KUKA KRL program: EPS_2_251806_MH49A_A_20260212042248.src

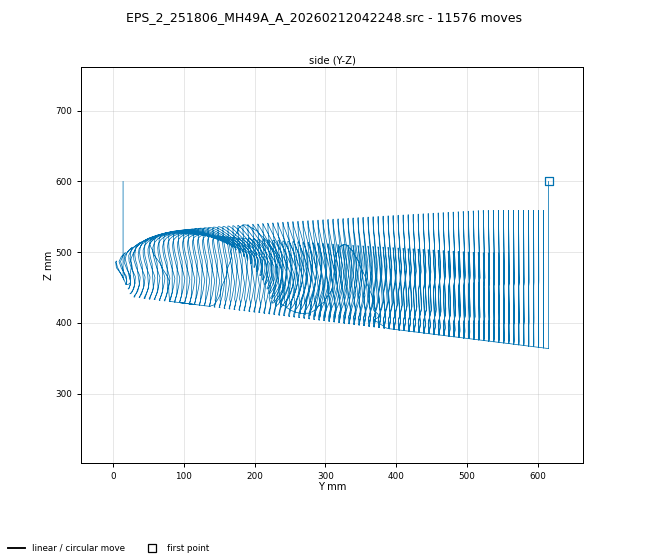
[picture p0: tool path of EPS_2_251806_MH49A_A_20260212042248.src, 11576 of 11578 moves have a stored position in this frame; points joined in program order, loops and branches not executed]
&ACCESS RVP
&REL 4
&COMMENT QRS 19112012
&PARAM EDITMASK = *
DEF PART()
EXT BAS (BAS_COMMAND :IN,REAL :IN )
INT I
BAS (#INITMOV,0 )

;KUKA QRS Post kuka4.cps  Date:22-06-2017 !

File_ID=3021

QRS_PRE_INIT()

;Init var - Until changes are made in qrs_pre_init
Outlet_Square_prg=0
Inlet_1_Square_prg=0
Inlet_2_Square_prg=0
Inlet_3_Square_prg=0
Inlet_4_Square_prg=0
Inlet_5_Square_prg=0

Outlet_1={X 0.000, Y 520.860, Z 458.500, B 0.000, E1 0.000 }
Inlet_1={X 0.000, Y 525.210, Z 398.500, B 0.000, E1 242.000 }
Outlet_1_type=201
Inlet_1_type=201
;QRS#1=Sidecore dimensions
;QRS#2=200-8" PVC SDR 35
;QRS#3=200-8" PVC SDR 35
;QRS#4=
;QRS#5=
;QRS#6=
;QRS#7=
;QRS#8=
;QRS#9=12-08 PSX
;QRS#10=12-08 PSX
;QRS#11=
;QRS#12=
;QRS#13=
;QRS#14=
;QRS#15=
;QRS#16=1220x127x838 2,75'
;QRS#17=EPS Height
;QRS#18=559
;QRS#19=*
;QRS#20= UPDATED VERSION 22-06-2017
;QRS#21=*
Outlet_Square=0100
Inlet_1_Square=0100
Inlet_2_Square=0
Inlet_3_Square=0
Inlet_4_Square=0
Inlet_5_Square=0
Mill_Square=1
Outlet_Square_Prg=204
Inlet_1_Square_prg=204

QRS_INIT()

$ADVANCE=5

; T1
PTP {E1 173.627,E2 173.627}
PTP {X 0,Y 615.485,A -85,B 0,C 180,E1 173.627,E2 173.627,E3 0,E4 0,E5 0,E6 0}
QRS_SPEED_INIT()
LIN {X 0,Y 615.485,Z 600,A -85,B 0,C 180,E1 173.627,E2 173.627,E3 0,E4 0,E5 0,E6 0} C_VEL
LIN {X 0,Y 615.485,Z 373.874,A -85,B 0,C 180,E1 173.627,E2 173.627} C_VEL
LIN {X 0,Y 615.485,Z 365.7,A -85,B 0,C 180,E1 173.627,E2 173.627} C_VEL
LIN {X 0,Y 615.471,Z 363.7,A -85,B 0,C 180,E1 173.44,E2 173.44} C_VEL
LIN {X 0,Y 615.49,Z 363.695,A -85,B 0,C 180,E1 170.802,E2 170.802} C_VEL
LIN {X 0,Y 615.467,Z 363.7,A -85,B 0,C 180,E1 168.139,E2 168.139} C_VEL
LIN {X 0,Y 615.473,Z 363.699,A -85,B 0,C 180,E1 165.451,E2 165.451} C_VEL
LIN {X 0,Y 615.485,Z 363.697,A -85,B 0,C 180,E1 162.73,E2 162.73} C_VEL
LIN {X 0,Y 615.476,Z 363.7,A -85,B 0,C 180,E1 159.968,E2 159.968} C_VEL
LIN {X 0,Y 615.494,Z 363.699,A -85,B 0,C 180,E1 157.156,E2 157.156} C_VEL
LIN {X 0,Y 615.492,Z 363.7,A -85,B 0,C 180,E1 154.285,E2 154.285} C_VEL
LIN {X 0,Y 615.492,Z 363.695,A -85,B 0,C 180,E1 151.343,E2 151.343} C_VEL
LIN {X 0,Y 615.482,Z 363.702,A -85,B 0,C 180,E1 148.916,E2 148.916} C_VEL
LIN {X 0,Y 615.483,Z 363.7,A -85,B 0,C 180,E1 146.468,E2 146.468} C_VEL
LIN {X 0,Y 615.46,Z 363.7,A -85,B 0,C 180,E1 144.171,E2 144.171} C_VEL
LIN {X 0,Y 615.483,Z 363.696,A -85,B 0,C 180,E1 141.932,E2 141.932} C_VEL
LIN {X 0,Y 615.49,Z 363.697,A -85,B 0,C 180,E1 139.395,E2 139.395} C_VEL
LIN {X 0,Y 615.481,Z 363.7,A -85,B 0,C 180,E1 136.756,E2 136.756} C_VEL
LIN {X 0,Y 615.489,Z 363.697,A -85,B 0,C 180,E1 133.999,E2 133.999} C_VEL
LIN {X 0,Y 615.464,Z 363.699,A -85,B 0,C 180,E1 131.093,E2 131.093} C_VEL
LIN {X 0,Y 615.493,Z 363.701,A -85,B 0,C 180,E1 128.906,E2 128.906} C_VEL
LIN {X 0,Y 615.492,Z 363.694,A -85,B 0,C 180,E1 125.836,E2 125.836} C_VEL
LIN {X 0,Y 615.472,Z 363.7,A -85,B 0,C 180,E1 123.239,E2 123.239} C_VEL
LIN {X 0,Y 615.495,Z 363.699,A -85,B 0,C 180,E1 120.921,E2 120.921} C_VEL
LIN {X 0,Y 615.472,Z 363.7,A -85,B 0,C 180,E1 118.449,E2 118.449} C_VEL
LIN {X 0,Y 615.499,Z 363.698,A -85,B 0,C 180,E1 115.573,E2 115.573} C_VEL
LIN {X 0,Y 615.488,Z 363.701,A -85,B 0,C 180,E1 112.846,E2 112.846} C_VEL
LIN {X 0,Y 615.494,Z 363.699,A -85,B 0,C 180,E1 110.034,E2 110.034} C_VEL
LIN {X 0,Y 615.483,Z 363.7,A -85,B 0,C 180,E1 107.273,E2 107.273} C_VEL
LIN {X 0,Y 615.483,Z 363.699,A -85,B 0,C 180,E1 104.551,E2 104.551} C_VEL
LIN {X 0,Y 615.49,Z 363.697,A -85,B 0,C 180,E1 101.863,E2 101.863} C_VEL
LIN {X 0,Y 615.48,Z 363.7,A -85,B 0,C 180,E1 99.201,E2 99.201} C_VEL
LIN {X 0,Y 615.488,Z 363.699,A -85,B 0,C 180,E1 96.559,E2 96.559} C_VEL
LIN {X 0,Y 615.486,Z 363.701,A -85,B 0,C 180,E1 93.931,E2 93.931} C_VEL
LIN {X 0,Y 615.493,Z 363.701,A -85,B 0,C 180,E1 91.311,E2 91.311} C_VEL
LIN {X 0,Y 615.493,Z 363.701,A -85,B 0,C 180,E1 88.694,E2 88.694} C_VEL
LIN {X 0,Y 615.486,Z 363.701,A -85,B 0,C 180,E1 86.074,E2 86.074} C_VEL
LIN {X 0,Y 615.488,Z 363.7,A -85,B 0,C 180,E1 83.414,E2 83.414} C_VEL
LIN {X 0,Y 615.48,Z 363.7,A -85,B 0,C 180,E1 80.804,E2 80.804} C_VEL
LIN {X 0,Y 615.49,Z 363.697,A -85,B 0,C 180,E1 78.142,E2 78.142} C_VEL
LIN {X 0,Y 615.483,Z 363.699,A -85,B 0,C 180,E1 75.454,E2 75.454} C_VEL
LIN {X 0,Y 615.483,Z 363.7,A -85,B 0,C 180,E1 72.732,E2 72.732} C_VEL
LIN {X 0,Y 615.497,Z 363.699,A -85,B 0,C 180,E1 69.971,E2 69.971} C_VEL
LIN {X 0,Y 615.49,Z 363.701,A -85,B 0,C 180,E1 67.159,E2 67.159} C_VEL
LIN {X 0,Y 615.5,Z 363.695,A -85,B 0,C 180,E1 64.288,E2 64.288} C_VEL
LIN {X 0,Y 615.475,Z 363.698,A -85,B 0,C 180,E1 63.559,E2 63.559} C_VEL
LIN {X 0,Y 615.495,Z 365.173,A -85,B 0,C 180,E1 62.089,E2 62.089} C_VEL
LIN {X 0,Y 615.491,Z 367.878,A -85,B 0,C 180,E1 59.844,E2 59.844} C_VEL
LIN {X 0,Y 615.43,Z 370.72,A -85,B 0,C 180,E1 57.543,E2 57.543} C_VEL
LIN {X 0,Y 615.447,Z 373.748,A -85,B 0,C 180,E1 55.187,E2 55.187} C_VEL
LIN {X 0,Y 615.494,Z 376.914,A -85,B 0,C 180,E1 52.763,E2 52.763} C_VEL
LIN {X 0,Y 615.478,Z 380.266,A -85,B 0,C 180,E1 50.254,E2 50.254} C_VEL
LIN {X 0,Y 615.456,Z 383.824,A -85,B 0,C 180,E1 47.649,E2 47.649} C_VEL
LIN {X 0,Y 615.491,Z 387.566,A -85,B 0,C 180,E1 44.937,E2 44.937} C_VEL
LIN {X 0,Y 615.483,Z 391.193,A -85,B 0,C 180,E1 42.352,E2 42.352} C_VEL
LIN {X 0,Y 615.485,Z 395.172,A -85,B 0,C 180,E1 39.557,E2 39.557} C_VEL
LIN {X 0,Y 615.487,Z 410.197,A -85,B 0,C 180,E1 39.195,E2 39.195} C_VEL
LIN {X 0,Y 615.486,Z 421.775,A -85,B 0,C 180,E1 38.798,E2 38.798} C_VEL
LIN {X 0,Y 615.479,Z 433.224,A -85,B 0,C 180,E1 38.276,E2 38.276} C_VEL
LIN {X 0,Y 615.485,Z 444.359,A -85,B 0,C 180,E1 37.628,E2 37.628} C_VEL
LIN {X 0,Y 615.495,Z 455.5,A -85,B 0,C 180,E1 36.813,E2 36.813} C_VEL
LIN {X 0,Y 615.497,Z 464.562,A -85,B 0,C 180,E1 35.987,E2 35.987} C_VEL
LIN {X 0,Y 615.496,Z 473.257,A -85,B 0,C 180,E1 35.013,E2 35.013} C_VEL
LIN {X 0,Y 615.496,Z 480.4,A -85,B 0,C 180,E1 34.02,E2 34.02} C_VEL
LIN {X 0,Y 615.495,Z 484.993,A -85,B 0,C 180,E1 33.235,E2 33.235} C_VEL
LIN {X 0,Y 615.493,Z 490.665,A -85,B 0,C 180,E1 32.011,E2 32.011} C_VEL
LIN {X 0,Y 615.497,Z 494.309,A -85,B 0,C 180,E1 30.918,E2 30.918} C_VEL
LIN {X 0,Y 615.496,Z 496.798,A -85,B 0,C 180,E1 29.804,E2 29.804} C_VEL
LIN {X 0,Y 615.498,Z 498.271,A -85,B 0,C 180,E1 28.46,E2 28.46} C_VEL
LIN {X 0,Y 615.494,Z 498.086,A -85,B 0,C 180,E1 27.176,E2 27.176} C_VEL
LIN {X 0,Y 615.494,Z 497.341,A -85,B 0,C 180,E1 26.443,E2 26.443} C_VEL
LIN {X 0,Y 615.494,Z 495.77,A -85,B 0,C 180,E1 25.579,E2 25.579} C_VEL
LIN {X 0,Y 615.497,Z 493.232,A -85,B 0,C 180,E1 24.63,E2 24.63} C_VEL
LIN {X 0,Y 615.496,Z 489.234,A -85,B 0,C 180,E1 23.555,E2 23.555} C_VEL
LIN {X 0,Y 615.497,Z 484.585,A -85,B 0,C 180,E1 22.601,E2 22.601} C_VEL
LIN {X 0,Y 615.495,Z 478.498,A -85,B 0,C 180,E1 21.607,E2 21.607} C_VEL
LIN {X 0,Y 615.497,Z 470.576,A -85,B 0,C 180,E1 20.571,E2 20.571} C_VEL
LIN {X 0,Y 615.497,Z 462.114,A -85,B 0,C 180,E1 19.684,E2 19.684} C_VEL
LIN {X 0,Y 615.498,Z 451.957,A -85,B 0,C 180,E1 18.818,E2 18.818} C_VEL
LIN {X 0,Y 615.466,Z 441.9,A -85,B 0,C 180,E1 18.123,E2 18.123} C_VEL
LIN {X 0,Y 615.442,Z 431.146,A -85,B 0,C 180,E1 17.528,E2 17.528} C_VEL
LIN {X 0,Y 615.475,Z 419.159,A -85,B 0,C 180,E1 17.013,E2 17.013} C_VEL
LIN {X 0,Y 615.495,Z 407.03,A -85,B 0,C 180,E1 16.628,E2 16.628} C_VEL
LIN {X 0,Y 615.481,Z 395.183,A -85,B 0,C 180,E1 16.36,E2 16.36} C_VEL
LIN {X 0,Y 615.433,Z 391.656,A -85,B 0,C 180,E1 13.875,E2 13.875} C_VEL
LIN {X 0,Y 615.426,Z 388.822,A -85,B 0,C 180,E1 11.861,E2 11.861} C_VEL
LIN {X 0,Y 615.419,Z 386.037,A -85,B 0,C 180,E1 9.863,E2 9.863} C_VEL
LIN {X 0,Y 615.458,Z 382.388,A -85,B 0,C 180,E1 7.215,E2 7.215} C_VEL
LIN {X 0,Y 615.451,Z 378.841,A -85,B 0,C 180,E1 4.584,E2 4.584} C_VEL
LIN {X 0,Y 615.429,Z 375.361,A -85,B 0,C 180,E1 1.963,E2 1.963} C_VEL
LIN {X 0,Y 615.485,Z 371.96,A -85,B 0,C 180,E1 -0.655,E2 -0.655} C_VEL
LIN {X 0,Y 615.485,Z 368.687,A -85,B 0,C 180,E1 -3.274,E2 -3.274} C_VEL
LIN {X 0,Y 615.496,Z 365.603,A -85,B 0,C 180,E1 -5.899,E2 -5.899} C_VEL
LIN {X 0,Y 615.493,Z 364.011,A -85,B 0,C 180,E1 -7.216,E2 -7.216} C_VEL
LIN {X 0,Y 615.468,Z 363.7,A -85,B 0,C 180,E1 -8.537,E2 -8.537} C_VEL
LIN {X 0,Y 615.482,Z 363.693,A -85,B 0,C 180,E1 -11.194,E2 -11.194} C_VEL
LIN {X 0,Y 615.448,Z 363.7,A -85,B 0,C 180,E1 -13.935,E2 -13.935} C_VEL
LIN {X 0,Y 615.493,Z 363.693,A -85,B 0,C 180,E1 -16.587,E2 -16.587} C_VEL
LIN {X 0,Y 615.482,Z 363.7,A -85,B 0,C 180,E1 -19.339,E2 -19.339} C_VEL
LIN {X 0,Y 615.49,Z 363.701,A -85,B 0,C 180,E1 -22.137,E2 -22.137} C_VEL
LIN {X 0,Y 615.496,Z 363.697,A -85,B 0,C 180,E1 -24.992,E2 -24.992} C_VEL
LIN {X 0,Y 615.48,Z 363.7,A -85,B 0,C 180,E1 -27.916,E2 -27.916} C_VEL
LIN {X 0,Y 615.472,Z 363.695,A -85,B 0,C 180,E1 -30.161,E2 -30.161} C_VEL
LIN {X 0,Y 615.482,Z 363.702,A -85,B 0,C 180,E1 -32.458,E2 -32.458} C_VEL
LIN {X 0,Y 615.484,Z 363.692,A -85,B 0,C 180,E1 -34.816,E2 -34.816} C_VEL
LIN {X 0,Y 615.471,Z 363.7,A -85,B 0,C 180,E1 -37.244,E2 -37.244} C_VEL
LIN {X 0,Y 615.494,Z 363.697,A -85,B 0,C 180,E1 -40.096,E2 -40.096} C_VEL
LIN {X 0,Y 615.485,Z 363.692,A -85,B 0,C 180,E1 -42.354,E2 -42.354} C_VEL
LIN {X 0,Y 615.457,Z 363.698,A -85,B 0,C 180,E1 -45.072,E2 -45.072} C_VEL
LIN {X 0,Y 615.479,Z 363.698,A -85,B 0,C 180,E1 -47.651,E2 -47.651} C_VEL
LIN {X 0,Y 615.49,Z 363.7,A -85,B 0,C 180,E1 -50.255,E2 -50.255} C_VEL
LIN {X 0,Y 615.481,Z 363.698,A -85,B 0,C 180,E1 -53.065,E2 -53.065} C_VEL
LIN {X 0,Y 615.492,Z 363.827,A -85,B 0,C 180,E1 -54.489,E2 -54.489} C_VEL
LIN {X 0,Y 615.488,Z 372.586,A -85,B 0,C 180,E1 -57.158,E2 -57.158} C_VEL
LIN {X 0,Y 615.445,Z 381.848,A -85,B 0,C 180,E1 -59.841,E2 -59.841} C_VEL
LIN {X 0,Y 615.439,Z 392.413,A -85,B 0,C 180,E1 -62.824,E2 -62.824} C_VEL
LIN {X 0,Y 615.439,Z 400.337,A -85,B 0,C 180,E1 -65.01,E2 -65.01} C_VEL
LIN {X 0,Y 615.484,Z 410.095,A -85,B 0,C 180,E1 -67.656,E2 -67.656} C_VEL
LIN {X 0,Y 615.486,Z 420.115,A -85,B 0,C 180,E1 -70.318,E2 -70.318} C_VEL
LIN {X 0,Y 615.487,Z 430.652,A -85,B 0,C 180,E1 -73.075,E2 -73.075} C_VEL
LIN {X 0,Y 615.472,Z 441.073,A -85,B 0,C 180,E1 -75.76,E2 -75.76} C_VEL
LIN {X 0,Y 615.494,Z 451.22,A -85,B 0,C 180,E1 -78.351,E2 -78.351} C_VEL
LIN {X 0,Y 615.499,Z 464.186,A -85,B 0,C 180,E1 -78.601,E2 -78.601} C_VEL
LIN {X 0,Y 615.463,Z 476.775,A -85,B 0,C 180,E1 -78.97,E2 -78.97} C_VEL
LIN {X 0,Y 615.45,Z 489.087,A -85,B 0,C 180,E1 -79.475,E2 -79.475} C_VEL
LIN {X 0,Y 615.486,Z 500.028,A -85,B 0,C 180,E1 -80.058,E2 -80.058} C_VEL
LIN {X 0,Y 615.499,Z 511.204,A -85,B 0,C 180,E1 -80.804,E2 -80.804} C_VEL
LIN {X 0,Y 615.498,Z 521.074,A -85,B 0,C 180,E1 -81.632,E2 -81.632} C_VEL
LIN {X 0,Y 615.498,Z 530.629,A -85,B 0,C 180,E1 -82.622,E2 -82.622} C_VEL
LIN {X 0,Y 615.496,Z 538.221,A -85,B 0,C 180,E1 -83.611,E2 -83.611} C_VEL
LIN {X 0,Y 615.498,Z 545.219,A -85,B 0,C 180,E1 -84.761,E2 -84.761} C_VEL
LIN {X 0,Y 615.494,Z 549.862,A -85,B 0,C 180,E1 -85.746,E2 -85.746} C_VEL
LIN {X 0,Y 615.494,Z 553.407,A -85,B 0,C 180,E1 -86.73,E2 -86.73} C_VEL
LIN {X 0,Y 615.497,Z 555.239,A -85,B 0,C 180,E1 -87.385,E2 -87.385} C_VEL
LIN {X 0,Y 615.499,Z 556.612,A -85,B 0,C 180,E1 -88.039,E2 -88.039} C_VEL
LIN {X 0,Y 615.496,Z 558.175,A -85,B 0,C 180,E1 -89.348,E2 -89.348} C_VEL
LIN {X 0,Y 615.494,Z 558.389,A -85,B 0,C 180,E1 -90.002,E2 -90.002} C_VEL
LIN {X 0,Y 615.495,Z 557.577,A -85,B 0,C 180,E1 -91.311,E2 -91.311} C_VEL
LIN {X 0,Y 615.499,Z 556.604,A -85,B 0,C 180,E1 -91.965,E2 -91.965} C_VEL
LIN {X 0,Y 615.497,Z 555.227,A -85,B 0,C 180,E1 -92.62,E2 -92.62} C_VEL
LIN {X 0,Y 615.496,Z 552.342,A -85,B 0,C 180,E1 -93.603,E2 -93.603} C_VEL
LIN {X 0,Y 615.498,Z 548.432,A -85,B 0,C 180,E1 -94.587,E2 -94.587} C_VEL
LIN {X 0,Y 615.499,Z 543.392,A -85,B 0,C 180,E1 -95.572,E2 -95.572} C_VEL
LIN {X 0,Y 615.497,Z 536.87,A -85,B 0,C 180,E1 -96.583,E2 -96.583} C_VEL
LIN {X 0,Y 615.497,Z 529.114,A -85,B 0,C 180,E1 -97.548,E2 -97.548} C_VEL
LIN {X 0,Y 615.498,Z 521.022,A -85,B 0,C 180,E1 -98.373,E2 -98.373} C_VEL
LIN {X 0,Y 615.499,Z 511.139,A -85,B 0,C 180,E1 -99.201,E2 -99.201} C_VEL
LIN {X 0,Y 615.487,Z 499.946,A -85,B 0,C 180,E1 -99.947,E2 -99.947} C_VEL
LIN {X 0,Y 615.449,Z 488.985,A -85,B 0,C 180,E1 -100.53,E2 -100.53} C_VEL
LIN {X 0,Y 615.463,Z 476.711,A -85,B 0,C 180,E1 -101.033,E2 -101.033} C_VEL
LIN {X 0,Y 615.499,Z 463.972,A -85,B 0,C 180,E1 -101.403,E2 -101.403} C_VEL
LIN {X 0,Y 615.494,Z 451.201,A -85,B 0,C 180,E1 -101.654,E2 -101.654} C_VEL
LIN {X 0,Y 615.472,Z 441.063,A -85,B 0,C 180,E1 -104.242,E2 -104.242} C_VEL
LIN {X 0,Y 615.487,Z 430.633,A -85,B 0,C 180,E1 -106.93,E2 -106.93} C_VEL
LIN {X 0,Y 615.484,Z 420.096,A -85,B 0,C 180,E1 -109.687,E2 -109.687} C_VEL
LIN {X 0,Y 615.484,Z 410.095,A -85,B 0,C 180,E1 -112.344,E2 -112.344} C_VEL
LIN {X 0,Y 615.439,Z 400.317,A -85,B 0,C 180,E1 -114.996,E2 -114.996} C_VEL
LIN {X 0,Y 615.478,Z 391.069,A -85,B 0,C 180,E1 -117.548,E2 -117.548} C_VEL
LIN {X 0,Y 615.445,Z 381.828,A -85,B 0,C 180,E1 -120.164,E2 -120.164} C_VEL
LIN {X 0,Y 615.488,Z 372.575,A -85,B 0,C 180,E1 -122.848,E2 -122.848} C_VEL
LIN {X 0,Y 615.495,Z 363.693,A -85,B 0,C 180,E1 -125.567,E2 -125.567} C_VEL
LIN {X 0,Y 615.476,Z 363.701,A -85,B 0,C 180,E1 -128.071,E2 -128.071} C_VEL
LIN {X 0,Y 615.49,Z 363.701,A -85,B 0,C 180,E1 -130.608,E2 -130.608} C_VEL
LIN {X 0,Y 615.5,Z 363.7,A -85,B 0,C 180,E1 -133.245,E2 -133.245} C_VEL
LIN {X 0,Y 615.487,Z 363.701,A -85,B 0,C 180,E1 -136.004,E2 -136.004} C_VEL
LIN {X 0,Y 615.483,Z 363.697,A -85,B 0,C 180,E1 -138.908,E2 -138.908} C_VEL
LIN {X 0,Y 615.475,Z 363.701,A -85,B 0,C 180,E1 -141.094,E2 -141.094} C_VEL
LIN {X 0,Y 615.49,Z 363.695,A -85,B 0,C 180,E1 -143.575,E2 -143.575} C_VEL
LIN {X 0,Y 615.48,Z 363.7,A -85,B 0,C 180,E1 -146.468,E2 -146.468} C_VEL
LIN {X 0,Y 615.475,Z 363.7,A -85,B 0,C 180,E1 -149.079,E2 -149.079} C_VEL
LIN {X 0,Y 615.49,Z 363.694,A -85,B 0,C 180,E1 -151.551,E2 -151.551} C_VEL
LIN {X 0,Y 615.475,Z 363.7,A -85,B 0,C 180,E1 -154.435,E2 -154.435} C_VEL
LIN {X 0,Y 615.489,Z 363.697,A -85,B 0,C 180,E1 -157.155,E2 -157.155} C_VEL
LIN {X 0,Y 615.486,Z 363.701,A -85,B 0,C 180,E1 -159.967,E2 -159.967} C_VEL
LIN {X 0,Y 615.496,Z 363.701,A -85,B 0,C 180,E1 -162.729,E2 -162.729} C_VEL
LIN {X 0,Y 615.488,Z 363.702,A -85,B 0,C 180,E1 -165.45,E2 -165.45} C_VEL
LIN {X 0,Y 615.487,Z 363.702,A -85,B 0,C 180,E1 -168.139,E2 -168.139} C_VEL
LIN {X 0,Y 615.499,Z 363.7,A -85,B 0,C 180,E1 -170.801,E2 -170.801} C_VEL
LIN {X 0,Y 615.493,Z 363.701,A -85,B 0,C 180,E1 -173.443,E2 -173.443} C_VEL
LIN {X 0,Y 615.486,Z 363.702,A -85,B 0,C 180,E1 -176.071,E2 -176.071} C_VEL
LIN {X 0,Y 615.483,Z 363.701,A -85,B 0,C 180,E1 -178.691,E2 -178.691} C_VEL
LIN {X 0,Y 615.494,Z 363.697,A -85,B 0,C 180,E1 -181.308,E2 -181.308} C_VEL
LIN {X 0,Y 615.477,Z 363.699,A -85,B 0,C 180,E1 -183.928,E2 -183.928} C_VEL
LIN {X 0,Y 615.471,Z 363.7,A -85,B 0,C 180,E1 -186.56,E2 -186.56} C_VEL
LIN {X 0,Y 614.8,Z 363.845,A -85,B 0,C 180,E1 -187.105,E2 -187.105} C_VEL
LIN {X 0,Y 611.979,Z 364.256,A -85,B 0,C 180,E1 -187.992,E2 -187.992} C_VEL
LIN {X 0,Y 609.593,Z 364.566,A -85,B 0,C 180,E1 -188.704,E2 -188.704} C_VEL
LIN {X 0,Y 608.552,Z 364.684,A -85,B 0,C 180,E1 -189.254,E2 -189.254} C_VEL
LIN {X 0,Y 608.458,Z 364.694,A -85,B 0,C 180,E1 -189.44,E2 -189.44} C_VEL
LIN {X 0,Y 608.45,Z 364.696,A -85,B 0,C 180,E1 -191.999,E2 -191.999} C_VEL
LIN {X 0,Y 608.435,Z 364.698,A -85,B 0,C 180,E1 -194.721,E2 -194.721} C_VEL
LIN {X 0,Y 608.449,Z 364.697,A -85,B 0,C 180,E1 -197.476,E2 -197.476} C_VEL
LIN {X 0,Y 608.461,Z 364.697,A -85,B 0,C 180,E1 -200.273,E2 -200.273} C_VEL
LIN {X 0,Y 608.445,Z 364.697,A -85,B 0,C 180,E1 -203.123,E2 -203.123} C_VEL
LIN {X 0,Y 608.478,Z 364.694,A -85,B 0,C 180,E1 -205.72,E2 -205.72} C_VEL
LIN {X 0,Y 608.481,Z 364.691,A -85,B 0,C 180,E1 -208.62,E2 -208.62} C_VEL
LIN {X 0,Y 608.444,Z 364.696,A -85,B 0,C 180,E1 -211.317,E2 -211.317} C_VEL
LIN {X 0,Y 608.476,Z 364.695,A -85,B 0,C 180,E1 -213.734,E2 -213.734} C_VEL
LIN {X 0,Y 608.444,Z 364.696,A -85,B 0,C 180,E1 -216.091,E2 -216.091} C_VEL
LIN {X 0,Y 608.474,Z 364.691,A -85,B 0,C 180,E1 -218.587,E2 -218.587} C_VEL
LIN {X 0,Y 608.45,Z 364.695,A -85,B 0,C 180,E1 -221.339,E2 -221.339} C_VEL
LIN {X 0,Y 608.454,Z 364.693,A -85,B 0,C 180,E1 -223.87,E2 -223.87} C_VEL
LIN {X 0,Y 608.479,Z 364.691,A -85,B 0,C 180,E1 -226.689,E2 -226.689} C_VEL
LIN {X 0,Y 608.455,Z 364.697,A -85,B 0,C 180,E1 -229.695,E2 -229.695} C_VEL
LIN {X 0,Y 608.453,Z 364.696,A -85,B 0,C 180,E1 -232.251,E2 -232.251} C_VEL
LIN {X 0,Y 608.484,Z 364.694,A -85,B 0,C 180,E1 -235.088,E2 -235.088} C_VEL
LIN {X 0,Y 608.467,Z 364.695,A -85,B 0,C 180,E1 -237.904,E2 -237.904} C_VEL
LIN {X 0,Y 608.471,Z 364.693,A -85,B 0,C 180,E1 -240.219,E2 -240.219} C_VEL
LIN {X 0,Y 608.445,Z 364.699,A -85,B 0,C 180,E1 -243.224,E2 -243.224} C_VEL
LIN {X 0,Y 608.485,Z 364.694,A -85,B 0,C 180,E1 -245.844,E2 -245.844} C_VEL
LIN {X 0,Y 608.472,Z 364.693,A -85,B 0,C 180,E1 -248.307,E2 -248.307} C_VEL
LIN {X 0,Y 608.47,Z 364.695,A -85,B 0,C 180,E1 -251.282,E2 -251.282} C_VEL
LIN {X 0,Y 608.459,Z 364.698,A -85,B 0,C 180,E1 -253.904,E2 -253.904} C_VEL
LIN {X 0,Y 608.461,Z 364.697,A -85,B 0,C 180,E1 -256.641,E2 -256.641} C_VEL
LIN {X 0,Y 608.465,Z 364.696,A -85,B 0,C 180,E1 -259.348,E2 -259.348} C_VEL
LIN {X 0,Y 608.476,Z 364.694,A -85,B 0,C 180,E1 -262.031,E2 -262.031} C_VEL
LIN {X 0,Y 608.466,Z 364.696,A -85,B 0,C 180,E1 -264.696,E2 -264.696} C_VEL
LIN {X 0,Y 608.479,Z 364.695,A -85,B 0,C 180,E1 -267.35,E2 -267.35} C_VEL
LIN {X 0,Y 608.472,Z 364.696,A -85,B 0,C 180,E1 -269.998,E2 -269.998} C_VEL
LIN {X 0,Y 608.479,Z 364.695,A -85,B 0,C 180,E1 -272.646,E2 -272.646} C_VEL
LIN {X 0,Y 608.466,Z 364.696,A -85,B 0,C 180,E1 -275.299,E2 -275.299} C_VEL
LIN {X 0,Y 608.475,Z 364.695,A -85,B 0,C 180,E1 -277.964,E2 -277.964} C_VEL
LIN {X 0,Y 608.462,Z 364.696,A -85,B 0,C 180,E1 -280.647,E2 -280.647} C_VEL
LIN {X 0,Y 608.46,Z 364.697,A -85,B 0,C 180,E1 -283.354,E2 -283.354} C_VEL
LIN {X 0,Y 608.458,Z 364.698,A -85,B 0,C 180,E1 -286.091,E2 -286.091} C_VEL
LIN {X 0,Y 608.446,Z 364.698,A -85,B 0,C 180,E1 -288.867,E2 -288.867} C_VEL
LIN {X 0,Y 608.47,Z 364.693,A -85,B 0,C 180,E1 -291.688,E2 -291.688} C_VEL
LIN {X 0,Y 608.44,Z 364.695,A -85,B 0,C 180,E1 -294.568,E2 -294.568} C_VEL
LIN {X 0,Y 608.414,Z 364.703,A -85,B 0,C 180,E1 -296.772,E2 -296.772} C_VEL
LIN {X 0,Y 608.438,Z 367.336,A -85,B 0,C 180,E1 -299.018,E2 -299.018} C_VEL
LIN {X 0,Y 608.429,Z 370.098,A -85,B 0,C 180,E1 -301.315,E2 -301.315} C_VEL
LIN {X 0,Y 608.417,Z 373.114,A -85,B 0,C 180,E1 -303.729,E2 -303.729} C_VEL
LIN {X 0,Y 608.418,Z 376.165,A -85,B 0,C 180,E1 -306.09,E2 -306.09} C_VEL
LIN {X 0,Y 608.389,Z 379.464,A -85,B 0,C 180,E1 -308.589,E2 -308.589} C_VEL
LIN {X 0,Y 608.429,Z 383.162,A -85,B 0,C 180,E1 -311.34,E2 -311.34} C_VEL
LIN {X 0,Y 608.399,Z 386.629,A -85,B 0,C 180,E1 -313.871,E2 -313.871} C_VEL
LIN {X 0,Y 608.431,Z 390.547,A -85,B 0,C 180,E1 -316.69,E2 -316.69} C_VEL
LIN {X 0,Y 608.421,Z 393.547,A -85,B 0,C 180,E1 -318.822,E2 -318.822} C_VEL
LIN {X 0,Y 608.425,Z 395.676,A -85,B 0,C 180,E1 -320.323,E2 -320.323} C_VEL
LIN {X 0,Y 608.529,Z 410.833,A -85,B 0,C 180,E1 -320.69,E2 -320.69} C_VEL
LIN {X 0,Y 608.511,Z 423.69,A -85,B 0,C 180,E1 -321.151,E2 -321.151} C_VEL
LIN {X 0,Y 608.489,Z 436.124,A -85,B 0,C 180,E1 -321.751,E2 -321.751} C_VEL
LIN {X 0,Y 608.502,Z 446.94,A -85,B 0,C 180,E1 -322.417,E2 -322.417} C_VEL
LIN {X 0,Y 608.483,Z 457.012,A -85,B 0,C 180,E1 -323.191,E2 -323.191} C_VEL
LIN {X 0,Y 608.471,Z 466.931,A -85,B 0,C 180,E1 -324.131,E2 -324.131} C_VEL
LIN {X 0,Y 608.46,Z 475.052,A -85,B 0,C 180,E1 -325.086,E2 -325.086} C_VEL
LIN {X 0,Y 608.436,Z 482.133,A -85,B 0,C 180,E1 -326.122,E2 -326.122} C_VEL
LIN {X 0,Y 608.431,Z 487.582,A -85,B 0,C 180,E1 -327.12,E2 -327.12} C_VEL
LIN {X 0,Y 608.437,Z 492.509,A -85,B 0,C 180,E1 -328.295,E2 -328.295} C_VEL
LIN {X 0,Y 608.448,Z 495.948,A -85,B 0,C 180,E1 -329.455,E2 -329.455} C_VEL
LIN {X 0,Y 608.443,Z 497.468,A -85,B 0,C 180,E1 -330.22,E2 -330.22} C_VEL
LIN {X 0,Y 608.424,Z 498.781,A -85,B 0,C 180,E1 -331.38,E2 -331.38} C_VEL
LIN {X 0,Y 608.429,Z 498.723,A -85,B 0,C 180,E1 -332.793,E2 -332.793} C_VEL
LIN {X 0,Y 608.416,Z 497.313,A -85,B 0,C 180,E1 -333.964,E2 -333.964} C_VEL
LIN {X 0,Y 608.43,Z 494.82,A -85,B 0,C 180,E1 -335.064,E2 -335.064} C_VEL
LIN {X 0,Y 608.438,Z 491.171,A -85,B 0,C 180,E1 -336.155,E2 -336.155} C_VEL
LIN {X 0,Y 608.459,Z 486.288,A -85,B 0,C 180,E1 -337.234,E2 -337.234} C_VEL
LIN {X 0,Y 608.459,Z 479.98,A -85,B 0,C 180,E1 -338.309,E2 -338.309} C_VEL
LIN {X 0,Y 608.466,Z 472.612,A -85,B 0,C 180,E1 -339.31,E2 -339.31} C_VEL
LIN {X 0,Y 608.473,Z 464.047,A -85,B 0,C 180,E1 -340.255,E2 -340.255} C_VEL
LIN {X 0,Y 608.482,Z 454.179,A -85,B 0,C 180,E1 -341.132,E2 -341.132} C_VEL
LIN {X 0,Y 608.479,Z 443.241,A -85,B 0,C 180,E1 -341.917,E2 -341.917} C_VEL
LIN {X 0,Y 608.467,Z 432.671,A -85,B 0,C 180,E1 -342.525,E2 -342.525} C_VEL
LIN {X 0,Y 608.49,Z 421.119,A -85,B 0,C 180,E1 -343.045,E2 -343.045} C_VEL
LIN {X 0,Y 608.555,Z 407.981,A -85,B 0,C 180,E1 -343.479,E2 -343.479} C_VEL
LIN {X 0,Y 608.399,Z 395.674,A -85,B 0,C 180,E1 -343.769,E2 -343.769} C_VEL
LIN {X 0,Y 608.393,Z 391.611,A -85,B 0,C 180,E1 -346.643,E2 -346.643} C_VEL
LIN {X 0,Y 608.411,Z 387.831,A -85,B 0,C 180,E1 -349.35,E2 -349.35} C_VEL
LIN {X 0,Y 608.352,Z 384.143,A -85,B 0,C 180,E1 -352.032,E2 -352.032} C_VEL
LIN {X 0,Y 608.419,Z 380.534,A -85,B 0,C 180,E1 -354.698,E2 -354.698} C_VEL
LIN {X 0,Y 608.393,Z 377.015,A -85,B 0,C 180,E1 -357.352,E2 -357.352} C_VEL
LIN {X 0,Y 608.4,Z 374.428,A -85,B 0,C 180,E1 -359.339,E2 -359.339} C_VEL
LIN {X 0,Y 608.411,Z 371.053,A -85,B 0,C 180,E1 -361.987,E2 -361.987} C_VEL
LIN {X 0,Y 608.449,Z 367.957,A -85,B 0,C 180,E1 -364.638,E2 -364.638} C_VEL
LIN {X 0,Y 608.439,Z 364.777,A -85,B 0,C 180,E1 -367.3,E2 -367.3} C_VEL
LIN {X 0,Y 608.435,Z 364.696,A -85,B 0,C 180,E1 -369.978,E2 -369.978} C_VEL
LIN {X 0,Y 608.466,Z 364.691,A -85,B 0,C 180,E1 -372.678,E2 -372.678} C_VEL
LIN {X 0,Y 608.445,Z 364.693,A -85,B 0,C 180,E1 -375.407,E2 -375.407} C_VEL
LIN {X 0,Y 608.444,Z 364.696,A -85,B 0,C 180,E1 -377.477,E2 -377.477} C_VEL
LIN {X 0,Y 608.434,Z 364.696,A -85,B 0,C 180,E1 -379.572,E2 -379.572} C_VEL
LIN {X 0,Y 608.464,Z 364.693,A -85,B 0,C 180,E1 -382.488,E2 -382.488} C_VEL
LIN {X 0,Y 608.439,Z 364.698,A -85,B 0,C 180,E1 -385.302,E2 -385.302} C_VEL
LIN {X 0,Y 608.45,Z 364.696,A -85,B 0,C 180,E1 -388.267,E2 -388.267} C_VEL
LIN {X 0,Y 608.464,Z 364.691,A -85,B 0,C 180,E1 -390.546,E2 -390.546} C_VEL
LIN {X 0,Y 608.436,Z 364.696,A -85,B 0,C 180,E1 -392.881,E2 -392.881} C_VEL
LIN {X 0,Y 608.445,Z 364.696,A -85,B 0,C 180,E1 -395.278,E2 -395.278} C_VEL
LIN {X 0,Y 608.444,Z 364.693,A -85,B 0,C 180,E1 -397.749,E2 -397.749} C_VEL
LIN {X 0,Y 608.458,Z 364.693,A -85,B 0,C 180,E1 -400.336,E2 -400.336} C_VEL
LIN {X 0,Y 608.452,Z 364.694,A -85,B 0,C 180,E1 -403.313,E2 -403.313} C_VEL
LIN {X 0,Y 608.475,Z 364.692,A -85,B 0,C 180,E1 -406.136,E2 -406.136} C_VEL
LIN {X 0,Y 608.455,Z 364.698,A -85,B 0,C 180,E1 -408.828,E2 -408.828} C_VEL
LIN {X 0,Y 608.465,Z 364.696,A -85,B 0,C 180,E1 -411.76,E2 -411.76} C_VEL
LIN {X 0,Y 608.507,Z 364.833,A -85,B 0,C 180,E1 -414.325,E2 -414.325} C_VEL
LIN {X 0,Y 608.523,Z 372.572,A -85,B 0,C 180,E1 -416.734,E2 -416.734} C_VEL
LIN {X 0,Y 608.481,Z 381.874,A -85,B 0,C 180,E1 -419.46,E2 -419.46} C_VEL
LIN {X 0,Y 608.485,Z 391.14,A -85,B 0,C 180,E1 -422.114,E2 -422.114} C_VEL
LIN {X 0,Y 608.443,Z 400.407,A -85,B 0,C 180,E1 -424.702,E2 -424.702} C_VEL
LIN {X 0,Y 608.437,Z 409.676,A -85,B 0,C 180,E1 -427.239,E2 -427.239} C_VEL
LIN {X 0,Y 608.465,Z 418.941,A -85,B 0,C 180,E1 -429.729,E2 -429.729} C_VEL
LIN {X 0,Y 608.455,Z 429.532,A -85,B 0,C 180,E1 -432.527,E2 -432.527} C_VEL
LIN {X 0,Y 608.439,Z 440.123,A -85,B 0,C 180,E1 -435.282,E2 -435.282} C_VEL
LIN {X 0,Y 608.426,Z 450.714,A -85,B 0,C 180,E1 -438.002,E2 -438.002} C_VEL
LIN {X 0,Y 608.441,Z 451.583,A -85,B 0,C 180,E1 -438.225,E2 -438.225} C_VEL
LIN {X 0,Y 608.567,Z 465.215,A -85,B 0,C 180,E1 -438.491,E2 -438.491} C_VEL
LIN {X 0,Y 608.488,Z 478.526,A -85,B 0,C 180,E1 -438.903,E2 -438.903} C_VEL
LIN {X 0,Y 608.478,Z 490.98,A -85,B 0,C 180,E1 -439.437,E2 -439.437} C_VEL
LIN {X 0,Y 608.486,Z 501.626,A -85,B 0,C 180,E1 -440.026,E2 -440.026} C_VEL
LIN {X 0,Y 608.483,Z 512.509,A -85,B 0,C 180,E1 -440.781,E2 -440.781} C_VEL
LIN {X 0,Y 608.474,Z 523.141,A -85,B 0,C 180,E1 -441.701,E2 -441.701} C_VEL
LIN {X 0,Y 608.47,Z 530.983,A -85,B 0,C 180,E1 -442.537,E2 -442.537} C_VEL
LIN {X 0,Y 608.459,Z 538.297,A -85,B 0,C 180,E1 -443.486,E2 -443.486} C_VEL
LIN {X 0,Y 608.45,Z 543.88,A -85,B 0,C 180,E1 -444.368,E2 -444.368} C_VEL
LIN {X 0,Y 608.432,Z 548.961,A -85,B 0,C 180,E1 -445.365,E2 -445.365} C_VEL
LIN {X 0,Y 608.449,Z 552.905,A -85,B 0,C 180,E1 -446.36,E2 -446.36} C_VEL
LIN {X 0,Y 608.425,Z 555.815,A -85,B 0,C 180,E1 -447.354,E2 -447.354} C_VEL
LIN {X 0,Y 608.444,Z 557.206,A -85,B 0,C 180,E1 -448.017,E2 -448.017} C_VEL
LIN {X 0,Y 608.438,Z 558.785,A -85,B 0,C 180,E1 -449.341,E2 -449.341} C_VEL
LIN {X 0,Y 608.434,Z 559,A -85,B 0,C 180,E1 -450.002,E2 -450.002} C_VEL
LIN {X 0,Y 608.448,Z 558.181,A -85,B 0,C 180,E1 -451.326,E2 -451.326} C_VEL
LIN {X 0,Y 608.444,Z 557.197,A -85,B 0,C 180,E1 -451.988,E2 -451.988} C_VEL
LIN {X 0,Y 608.425,Z 555.803,A -85,B 0,C 180,E1 -452.651,E2 -452.651} C_VEL
LIN {X 0,Y 608.449,Z 552.888,A -85,B 0,C 180,E1 -453.645,E2 -453.645} C_VEL
LIN {X 0,Y 608.432,Z 548.94,A -85,B 0,C 180,E1 -454.64,E2 -454.64} C_VEL
LIN {X 0,Y 608.437,Z 542.863,A -85,B 0,C 180,E1 -455.803,E2 -455.803} C_VEL
LIN {X 0,Y 608.464,Z 536.218,A -85,B 0,C 180,E1 -456.802,E2 -456.802} C_VEL
LIN {X 0,Y 608.456,Z 527.969,A -85,B 0,C 180,E1 -457.802,E2 -457.802} C_VEL
LIN {X 0,Y 608.472,Z 519.511,A -85,B 0,C 180,E1 -458.638,E2 -458.638} C_VEL
LIN {X 0,Y 608.481,Z 509.061,A -85,B 0,C 180,E1 -459.475,E2 -459.475} C_VEL
LIN {X 0,Y 608.499,Z 498.72,A -85,B 0,C 180,E1 -460.147,E2 -460.147} C_VEL
LIN {X 0,Y 608.473,Z 487.802,A -85,B 0,C 180,E1 -460.716,E2 -460.716} C_VEL
LIN {X 0,Y 608.496,Z 476.016,A -85,B 0,C 180,E1 -461.189,E2 -461.189} C_VEL
LIN {X 0,Y 608.55,Z 463.176,A -85,B 0,C 180,E1 -461.557,E2 -461.557} C_VEL
LIN {X 0,Y 608.445,Z 451.522,A -85,B 0,C 180,E1 -461.791,E2 -461.791} C_VEL
LIN {X 0,Y 608.437,Z 441.428,A -85,B 0,C 180,E1 -464.382,E2 -464.382} C_VEL
LIN {X 0,Y 608.444,Z 430.837,A -85,B 0,C 180,E1 -467.132,E2 -467.132} C_VEL
LIN {X 0,Y 608.454,Z 421.57,A -85,B 0,C 180,E1 -469.572,E2 -469.572} C_VEL
LIN {X 0,Y 608.47,Z 410.718,A -85,B 0,C 180,E1 -472.478,E2 -472.478} C_VEL
LIN {X 0,Y 608.43,Z 401.712,A -85,B 0,C 180,E1 -474.938,E2 -474.938} C_VEL
LIN {X 0,Y 608.473,Z 392.445,A -85,B 0,C 180,E1 -477.519,E2 -477.519} C_VEL
LIN {X 0,Y 608.48,Z 383.835,A -85,B 0,C 180,E1 -479.973,E2 -479.973} C_VEL
LIN {X 0,Y 608.523,Z 375.066,A -85,B 0,C 180,E1 -482.531,E2 -482.531} C_VEL
LIN {X 0,Y 608.557,Z 366.021,A -85,B 0,C 180,E1 -485.272,E2 -485.272} C_VEL
LIN {X 0,Y 608.466,Z 364.693,A -85,B 0,C 180,E1 -485.729,E2 -485.729} C_VEL
LIN {X 0,Y 608.46,Z 364.693,A -85,B 0,C 180,E1 -488.239,E2 -488.239} C_VEL
LIN {X 0,Y 608.448,Z 364.694,A -85,B 0,C 180,E1 -491.179,E2 -491.179} C_VEL
LIN {X 0,Y 608.465,Z 364.692,A -85,B 0,C 180,E1 -493.871,E2 -493.871} C_VEL
LIN {X 0,Y 608.453,Z 364.693,A -85,B 0,C 180,E1 -496.694,E2 -496.694} C_VEL
LIN {X 0,Y 608.464,Z 364.694,A -85,B 0,C 180,E1 -499.697,E2 -499.697} C_VEL
LIN {X 0,Y 608.479,Z 364.692,A -85,B 0,C 180,E1 -502.842,E2 -502.842} C_VEL
LIN {X 0,Y 608.468,Z 364.694,A -85,B 0,C 180,E1 -505.53,E2 -505.53} C_VEL
LIN {X 0,Y 608.465,Z 364.696,A -85,B 0,C 180,E1 -507.905,E2 -507.905} C_VEL
LIN {X 0,Y 608.474,Z 364.692,A -85,B 0,C 180,E1 -510.98,E2 -510.98} C_VEL
LIN {X 0,Y 608.432,Z 364.696,A -85,B 0,C 180,E1 -513.963,E2 -513.963} C_VEL
LIN {X 0,Y 608.465,Z 364.695,A -85,B 0,C 180,E1 -516.155,E2 -516.155} C_VEL
LIN {X 0,Y 608.462,Z 364.694,A -85,B 0,C 180,E1 -519.018,E2 -519.018} C_VEL
LIN {X 0,Y 608.432,Z 364.696,A -85,B 0,C 180,E1 -521.827,E2 -521.827} C_VEL
LIN {X 0,Y 608.462,Z 364.692,A -85,B 0,C 180,E1 -524.593,E2 -524.593} C_VEL
LIN {X 0,Y 608.475,Z 364.691,A -85,B 0,C 180,E1 -527.323,E2 -527.323} C_VEL
LIN {X 0,Y 608.436,Z 364.695,A -85,B 0,C 180,E1 -530.022,E2 -530.022} C_VEL
LIN {X 0,Y 608.449,Z 364.694,A -85,B 0,C 180,E1 -532.7,E2 -532.7} C_VEL
LIN {X 0,Y 608.443,Z 364.695,A -85,B 0,C 180,E1 -535.362,E2 -535.362} C_VEL
LIN {X 0,Y 608.487,Z 364.692,A -85,B 0,C 180,E1 -537.351,E2 -537.351} C_VEL
LIN {X 0,Y 608.477,Z 364.693,A -85,B 0,C 180,E1 -539.999,E2 -539.999} C_VEL
LIN {X 0,Y 608.467,Z 364.694,A -85,B 0,C 180,E1 -542.647,E2 -542.647} C_VEL
LIN {X 0,Y 608.469,Z 364.694,A -85,B 0,C 180,E1 -545.301,E2 -545.301} C_VEL
LIN {X 0,Y 608.44,Z 364.697,A -85,B 0,C 180,E1 -547.967,E2 -547.967} C_VEL
LIN {X 0,Y 608.458,Z 364.694,A -85,B 0,C 180,E1 -549.44,E2 -549.44} C_VEL
LIN {X 0,Y 607.767,Z 364.78,A -85,B 0,C 180,E1 -549.992,E2 -549.992} C_VEL
LIN {X 0,Y 604.909,Z 365.14,A -85,B 0,C 180,E1 -550.889,E2 -550.889} C_VEL
LIN {X 0,Y 602.512,Z 365.439,A -85,B 0,C 180,E1 -551.61,E2 -551.61} C_VEL
LIN {X 0,Y 601.487,Z 365.565,A -85,B 0,C 180,E1 -552.167,E2 -552.167} C_VEL
LIN {X 0,Y 601.405,Z 365.573,A -85,B 0,C 180,E1 -552.355,E2 -552.355} C_VEL
LIN {X 0,Y 601.402,Z 365.577,A -85,B 0,C 180,E1 -554.897,E2 -554.897} C_VEL
LIN {X 0,Y 601.435,Z 365.568,A -85,B 0,C 180,E1 -556.985,E2 -556.985} C_VEL
LIN {X 0,Y 601.398,Z 365.572,A -85,B 0,C 180,E1 -559.809,E2 -559.809} C_VEL
LIN {X 0,Y 601.401,Z 365.573,A -85,B 0,C 180,E1 -561.959,E2 -561.959} C_VEL
LIN {X 0,Y 601.404,Z 365.571,A -85,B 0,C 180,E1 -564.878,E2 -564.878} C_VEL
LIN {X 0,Y 601.401,Z 365.573,A -85,B 0,C 180,E1 -567.358,E2 -567.358} C_VEL
LIN {X 0,Y 601.423,Z 365.571,A -85,B 0,C 180,E1 -569.392,E2 -569.392} C_VEL
LIN {X 0,Y 601.44,Z 365.57,A -85,B 0,C 180,E1 -572.514,E2 -572.514} C_VEL
LIN {X 0,Y 601.396,Z 365.576,A -85,B 0,C 180,E1 -575.11,E2 -575.11} C_VEL
LIN {X 0,Y 601.435,Z 365.569,A -85,B 0,C 180,E1 -577.418,E2 -577.418} C_VEL
LIN {X 0,Y 601.401,Z 365.572,A -85,B 0,C 180,E1 -579.995,E2 -579.995} C_VEL
LIN {X 0,Y 601.415,Z 365.571,A -85,B 0,C 180,E1 -582.669,E2 -582.669} C_VEL
LIN {X 0,Y 601.401,Z 365.574,A -85,B 0,C 180,E1 -585.478,E2 -585.478} C_VEL
LIN {X 0,Y 601.416,Z 365.575,A -85,B 0,C 180,E1 -588.406,E2 -588.406} C_VEL
LIN {X 0,Y 601.432,Z 365.57,A -85,B 0,C 180,E1 -590.873,E2 -590.873} C_VEL
LIN {X 0,Y 601.406,Z 365.575,A -85,B 0,C 180,E1 -593.737,E2 -593.737} C_VEL
LIN {X 0,Y 601.433,Z 365.568,A -85,B 0,C 180,E1 -596.063,E2 -596.063} C_VEL
LIN {X 0,Y 601.423,Z 365.573,A -85,B 0,C 180,E1 -599.056,E2 -599.056} C_VEL
LIN {X 0,Y 601.42,Z 365.571,A -85,B 0,C 180,E1 -602.131,E2 -602.131} C_VEL
LIN {X 0,Y 601.395,Z 365.572,A -85,B 0,C 180,E1 -605.119,E2 -605.119} C_VEL
LIN {X 0,Y 601.415,Z 365.573,A -85,B 0,C 180,E1 -607.392,E2 -607.392} C_VEL
LIN {X 0,Y 601.402,Z 365.573,A -85,B 0,C 180,E1 -610.188,E2 -610.188} C_VEL
LIN {X 0,Y 601.408,Z 365.571,A -85,B 0,C 180,E1 -613.011,E2 -613.011} C_VEL
LIN {X 0,Y 601.42,Z 365.569,A -85,B 0,C 180,E1 -615.905,E2 -615.905} C_VEL
LIN {X 0,Y 601.426,Z 365.57,A -85,B 0,C 180,E1 -618.983,E2 -618.983} C_VEL
LIN {X 0,Y 601.436,Z 365.572,A -85,B 0,C 180,E1 -621.937,E2 -621.937} C_VEL
LIN {X 0,Y 601.432,Z 365.573,A -85,B 0,C 180,E1 -624.634,E2 -624.634} C_VEL
LIN {X 0,Y 601.443,Z 365.571,A -85,B 0,C 180,E1 -627.319,E2 -627.319} C_VEL
LIN {X 0,Y 601.44,Z 365.572,A -85,B 0,C 180,E1 -629.998,E2 -629.998} C_VEL
LIN {X 0,Y 601.442,Z 365.571,A -85,B 0,C 180,E1 -632.676,E2 -632.676} C_VEL
LIN {X 0,Y 601.432,Z 365.573,A -85,B 0,C 180,E1 -635.361,E2 -635.361} C_VEL
LIN {X 0,Y 601.434,Z 365.572,A -85,B 0,C 180,E1 -638.058,E2 -638.058} C_VEL
LIN {X 0,Y 601.421,Z 365.571,A -85,B 0,C 180,E1 -641.014,E2 -641.014} C_VEL
LIN {X 0,Y 601.41,Z 365.571,A -85,B 0,C 180,E1 -644.091,E2 -644.091} C_VEL
LIN {X 0,Y 601.418,Z 365.57,A -85,B 0,C 180,E1 -646.983,E2 -646.983} C_VEL
LIN {X 0,Y 601.4,Z 365.573,A -85,B 0,C 180,E1 -649.806,E2 -649.806} C_VEL
LIN {X 0,Y 601.418,Z 365.573,A -85,B 0,C 180,E1 -652.679,E2 -652.679} C_VEL
LIN {X 0,Y 601.391,Z 365.573,A -85,B 0,C 180,E1 -654.876,E2 -654.876} C_VEL
LIN {X 0,Y 601.372,Z 365.648,A -85,B 0,C 180,E1 -657.111,E2 -657.111} C_VEL
LIN {X 0,Y 601.383,Z 369.28,A -85,B 0,C 180,E1 -660.163,E2 -660.163} C_VEL
LIN {X 0,Y 601.314,Z 372.321,A -85,B 0,C 180,E1 -662.701,E2 -662.701} C_VEL
LIN {X 0,Y 601.325,Z 375.322,A -85,B 0,C 180,E1 -665.104,E2 -665.104} C_VEL
LIN {X 0,Y 601.336,Z 378.317,A -85,B 0,C 180,E1 -667.422,E2 -667.422} C_VEL
LIN {X 0,Y 601.323,Z 381.712,A -85,B 0,C 180,E1 -669.997,E2 -669.997} C_VEL
LIN {X 0,Y 601.348,Z 385.299,A -85,B 0,C 180,E1 -672.671,E2 -672.671} C_VEL
LIN {X 0,Y 601.329,Z 389.127,A -85,B 0,C 180,E1 -675.474,E2 -675.474} C_VEL
LIN {X 0,Y 601.304,Z 392.938,A -85,B 0,C 180,E1 -678.226,E2 -678.226} C_VEL
LIN {X 0,Y 601.325,Z 395.679,A -85,B 0,C 180,E1 -680.185,E2 -680.185} C_VEL
LIN {X 0,Y 601.606,Z 404.342,A -85,B 0,C 180,E1 -680.38,E2 -680.38} C_VEL
LIN {X 0,Y 601.568,Z 417.02,A -85,B 0,C 180,E1 -680.761,E2 -680.761} C_VEL
LIN {X 0,Y 601.538,Z 428.43,A -85,B 0,C 180,E1 -681.235,E2 -681.235} C_VEL
LIN {X 0,Y 601.476,Z 439.804,A -85,B 0,C 180,E1 -681.844,E2 -681.844} C_VEL
LIN {X 0,Y 601.472,Z 451.099,A -85,B 0,C 180,E1 -682.607,E2 -682.607} C_VEL
LIN {X 0,Y 601.444,Z 460.75,A -85,B 0,C 180,E1 -683.421,E2 -683.421} C_VEL
LIN {X 0,Y 601.39,Z 470.336,A -85,B 0,C 180,E1 -684.419,E2 -684.419} C_VEL
LIN {X 0,Y 601.386,Z 478.433,A -85,B 0,C 180,E1 -685.474,E2 -685.474} C_VEL
LIN {X 0,Y 601.377,Z 484.04,A -85,B 0,C 180,E1 -686.376,E2 -686.376} C_VEL
LIN {X 0,Y 601.334,Z 489.487,A -85,B 0,C 180,E1 -687.479,E2 -687.479} C_VEL
LIN {X 0,Y 601.352,Z 493.494,A -85,B 0,C 180,E1 -688.548,E2 -688.548} C_VEL
LIN {X 0,Y 601.351,Z 496.872,A -85,B 0,C 180,E1 -689.856,E2 -689.856} C_VEL
LIN {X 0,Y 601.334,Z 498.065,A -85,B 0,C 180,E1 -690.603,E2 -690.603} C_VEL
LIN {X 0,Y 601.331,Z 498.779,A -85,B 0,C 180,E1 -691.369,E2 -691.369} C_VEL
LIN {X 0,Y 601.34,Z 498.834,A -85,B 0,C 180,E1 -692.643,E2 -692.643} C_VEL
LIN {X 0,Y 601.309,Z 497.888,A -85,B 0,C 180,E1 -693.633,E2 -693.633} C_VEL
LIN {X 0,Y 601.326,Z 496.563,A -85,B 0,C 180,E1 -694.378,E2 -694.378} C_VEL
LIN {X 0,Y 601.355,Z 494.766,A -85,B 0,C 180,E1 -695.12,E2 -695.12} C_VEL
LIN {X 0,Y 601.369,Z 491.097,A -85,B 0,C 180,E1 -696.223,E2 -696.223} C_VEL
LIN {X 0,Y 601.354,Z 485.743,A -85,B 0,C 180,E1 -697.398,E2 -697.398} C_VEL
LIN {X 0,Y 601.384,Z 478.663,A -85,B 0,C 180,E1 -698.581,E2 -698.581} C_VEL
LIN {X 0,Y 601.4,Z 470.462,A -85,B 0,C 180,E1 -699.657,E2 -699.657} C_VEL
LIN {X 0,Y 601.434,Z 462.024,A -85,B 0,C 180,E1 -700.548,E2 -700.548} C_VEL
LIN {X 0,Y 601.471,Z 452.483,A -85,B 0,C 180,E1 -701.375,E2 -701.375} C_VEL
LIN {X 0,Y 601.439,Z 441.614,A -85,B 0,C 180,E1 -702.138,E2 -702.138} C_VEL
LIN {X 0,Y 601.468,Z 430.55,A -85,B 0,C 180,E1 -702.753,E2 -702.753} C_VEL
LIN {X 0,Y 601.535,Z 418.068,A -85,B 0,C 180,E1 -703.29,E2 -703.29} C_VEL
LIN {X 0,Y 601.581,Z 404.942,A -85,B 0,C 180,E1 -703.696,E2 -703.696} C_VEL
LIN {X 0,Y 601.476,Z 397.126,A -85,B 0,C 180,E1 -703.867,E2 -703.867} C_VEL
LIN {X 0,Y 601.299,Z 395.648,A -85,B 0,C 180,E1 -703.928,E2 -703.928} C_VEL
LIN {X 0,Y 601.29,Z 392.079,A -85,B 0,C 180,E1 -706.482,E2 -706.482} C_VEL
LIN {X 0,Y 601.317,Z 388.294,A -85,B 0,C 180,E1 -709.223,E2 -709.223} C_VEL
LIN {X 0,Y 601.271,Z 384.602,A -85,B 0,C 180,E1 -711.938,E2 -711.938} C_VEL
LIN {X 0,Y 601.323,Z 380.991,A -85,B 0,C 180,E1 -714.636,E2 -714.636} C_VEL
LIN {X 0,Y 601.305,Z 377.469,A -85,B 0,C 180,E1 -717.321,E2 -717.321} C_VEL
LIN {X 0,Y 601.324,Z 374.882,A -85,B 0,C 180,E1 -719.331,E2 -719.331} C_VEL
LIN {X 0,Y 601.343,Z 372.403,A -85,B 0,C 180,E1 -721.34,E2 -721.34} C_VEL
LIN {X 0,Y 601.38,Z 369.318,A -85,B 0,C 180,E1 -724.021,E2 -724.021} C_VEL
LIN {X 0,Y 601.392,Z 366.132,A -85,B 0,C 180,E1 -726.712,E2 -726.712} C_VEL
LIN {X 0,Y 601.393,Z 365.578,A -85,B 0,C 180,E1 -727.386,E2 -727.386} C_VEL
LIN {X 0,Y 601.416,Z 365.572,A -85,B 0,C 180,E1 -730.096,E2 -730.096} C_VEL
LIN {X 0,Y 601.413,Z 365.57,A -85,B 0,C 180,E1 -732.829,E2 -732.829} C_VEL
LIN {X 0,Y 601.392,Z 365.572,A -85,B 0,C 180,E1 -735.592,E2 -735.592} C_VEL
LIN {X 0,Y 601.391,Z 365.578,A -85,B 0,C 180,E1 -737.689,E2 -737.689} C_VEL
LIN {X 0,Y 601.415,Z 365.573,A -85,B 0,C 180,E1 -740.523,E2 -740.523} C_VEL
LIN {X 0,Y 601.414,Z 365.572,A -85,B 0,C 180,E1 -743.411,E2 -743.411} C_VEL
LIN {X 0,Y 601.381,Z 365.576,A -85,B 0,C 180,E1 -746.365,E2 -746.365} C_VEL
LIN {X 0,Y 601.433,Z 365.567,A -85,B 0,C 180,E1 -748.797,E2 -748.797} C_VEL
LIN {X 0,Y 601.415,Z 365.57,A -85,B 0,C 180,E1 -751.462,E2 -751.462} C_VEL
LIN {X 0,Y 601.416,Z 365.574,A -85,B 0,C 180,E1 -754.12,E2 -754.12} C_VEL
LIN {X 0,Y 601.405,Z 365.571,A -85,B 0,C 180,E1 -756.583,E2 -756.583} C_VEL
LIN {X 0,Y 601.422,Z 365.569,A -85,B 0,C 180,E1 -759.54,E2 -759.54} C_VEL
LIN {X 0,Y 601.412,Z 365.571,A -85,B 0,C 180,E1 -761.767,E2 -761.767} C_VEL
LIN {X 0,Y 601.4,Z 365.575,A -85,B 0,C 180,E1 -764.538,E2 -764.538} C_VEL
LIN {X 0,Y 601.421,Z 365.574,A -85,B 0,C 180,E1 -767.409,E2 -767.409} C_VEL
LIN {X 0,Y 601.424,Z 365.573,A -85,B 0,C 180,E1 -770.467,E2 -770.467} C_VEL
LIN {X 0,Y 601.403,Z 365.576,A -85,B 0,C 180,E1 -773.421,E2 -773.421} C_VEL
LIN {X 0,Y 601.436,Z 365.587,A -85,B 0,C 180,E1 -774.072,E2 -774.072} C_VEL
LIN {X 0,Y 601.579,Z 371.718,A -85,B 0,C 180,E1 -776.044,E2 -776.044} C_VEL
LIN {X 0,Y 601.517,Z 379.944,A -85,B 0,C 180,E1 -778.531,E2 -778.531} C_VEL
LIN {X 0,Y 601.457,Z 389.227,A -85,B 0,C 180,E1 -781.208,E2 -781.208} C_VEL
LIN {X 0,Y 601.485,Z 399.448,A -85,B 0,C 180,E1 -784.119,E2 -784.119} C_VEL
LIN {X 0,Y 601.405,Z 409.674,A -85,B 0,C 180,E1 -786.957,E2 -786.957} C_VEL
LIN {X 0,Y 601.43,Z 418.941,A -85,B 0,C 180,E1 -789.481,E2 -789.481} C_VEL
LIN {X 0,Y 601.402,Z 429.532,A -85,B 0,C 180,E1 -792.315,E2 -792.315} C_VEL
LIN {X 0,Y 601.367,Z 440.123,A -85,B 0,C 180,E1 -795.105,E2 -795.105} C_VEL
LIN {X 0,Y 601.352,Z 449.39,A -85,B 0,C 180,E1 -797.516,E2 -797.516} C_VEL
LIN {X 0,Y 601.383,Z 451.541,A -85,B 0,C 180,E1 -798.074,E2 -798.074} C_VEL
LIN {X 0,Y 601.611,Z 457.385,A -85,B 0,C 180,E1 -798.185,E2 -798.185} C_VEL
LIN {X 0,Y 601.559,Z 470.598,A -85,B 0,C 180,E1 -798.504,E2 -798.504} C_VEL
LIN {X 0,Y 601.501,Z 483.117,A -85,B 0,C 180,E1 -798.953,E2 -798.953} C_VEL
LIN {X 0,Y 601.474,Z 495.826,A -85,B 0,C 180,E1 -799.568,E2 -799.568} C_VEL
LIN {X 0,Y 601.473,Z 506.788,A -85,B 0,C 180,E1 -800.248,E2 -800.248} C_VEL
LIN {X 0,Y 601.434,Z 517.631,A -85,B 0,C 180,E1 -801.096,E2 -801.096} C_VEL
LIN {X 0,Y 601.406,Z 526.44,A -85,B 0,C 180,E1 -801.942,E2 -801.942} C_VEL
LIN {X 0,Y 601.382,Z 535.018,A -85,B 0,C 180,E1 -802.954,E2 -802.954} C_VEL
LIN {X 0,Y 601.36,Z 541.882,A -85,B 0,C 180,E1 -803.965,E2 -803.965} C_VEL
LIN {X 0,Y 601.345,Z 547.378,A -85,B 0,C 180,E1 -804.974,E2 -804.974} C_VEL
LIN {X 0,Y 601.346,Z 551.686,A -85,B 0,C 180,E1 -805.982,E2 -805.982} C_VEL
LIN {X 0,Y 601.344,Z 553.964,A -85,B 0,C 180,E1 -806.653,E2 -806.653} C_VEL
LIN {X 0,Y 601.325,Z 555.815,A -85,B 0,C 180,E1 -807.323,E2 -807.323} C_VEL
LIN {X 0,Y 601.343,Z 557.206,A -85,B 0,C 180,E1 -807.993,E2 -807.993} C_VEL
LIN {X 0,Y 601.339,Z 558.785,A -85,B 0,C 180,E1 -809.333,E2 -809.333} C_VEL
LIN {X 0,Y 601.335,Z 559,A -85,B 0,C 180,E1 -810.002,E2 -810.002} C_VEL
LIN {X 0,Y 601.348,Z 558.181,A -85,B 0,C 180,E1 -811.342,E2 -811.342} C_VEL
LIN {X 0,Y 601.343,Z 557.198,A -85,B 0,C 180,E1 -812.012,E2 -812.012} C_VEL
LIN {X 0,Y 601.325,Z 555.803,A -85,B 0,C 180,E1 -812.682,E2 -812.682} C_VEL
LIN {X 0,Y 601.368,Z 552.888,A -85,B 0,C 180,E1 -813.688,E2 -813.688} C_VEL
LIN {X 0,Y 601.336,Z 548.94,A -85,B 0,C 180,E1 -814.695,E2 -814.695} C_VEL
LIN {X 0,Y 601.372,Z 542.863,A -85,B 0,C 180,E1 -815.871,E2 -815.871} C_VEL
LIN {X 0,Y 601.384,Z 536.219,A -85,B 0,C 180,E1 -816.882,E2 -816.882} C_VEL
LIN {X 0,Y 601.401,Z 527.97,A -85,B 0,C 180,E1 -817.894,E2 -817.894} C_VEL
LIN {X 0,Y 601.437,Z 519.512,A -85,B 0,C 180,E1 -818.74,E2 -818.74} C_VEL
LIN {X 0,Y 601.451,Z 509.062,A -85,B 0,C 180,E1 -819.587,E2 -819.587} C_VEL
LIN {X 0,Y 601.489,Z 498.721,A -85,B 0,C 180,E1 -820.266,E2 -820.266} C_VEL
LIN {X 0,Y 601.488,Z 487.179,A -85,B 0,C 180,E1 -820.871,E2 -820.871} C_VEL
LIN {X 0,Y 601.529,Z 474.27,A -85,B 0,C 180,E1 -821.377,E2 -821.377} C_VEL
LIN {X 0,Y 601.602,Z 461.347,A -85,B 0,C 180,E1 -821.735,E2 -821.735} C_VEL
LIN {X 0,Y 601.412,Z 451.958,A -85,B 0,C 180,E1 -821.909,E2 -821.909} C_VEL
LIN {X 0,Y 601.357,Z 451.357,A -85,B 0,C 180,E1 -821.975,E2 -821.975} C_VEL
LIN {X 0,Y 601.387,Z 441.428,A -85,B 0,C 180,E1 -824.554,E2 -824.554} C_VEL
LIN {X 0,Y 601.39,Z 430.837,A -85,B 0,C 180,E1 -827.339,E2 -827.339} C_VEL
LIN {X 0,Y 601.429,Z 420.246,A -85,B 0,C 180,E1 -830.167,E2 -830.167} C_VEL
LIN {X 0,Y 601.416,Z 410.979,A -85,B 0,C 180,E1 -832.685,E2 -832.685} C_VEL
LIN {X 0,Y 601.43,Z 401.712,A -85,B 0,C 180,E1 -835.249,E2 -835.249} C_VEL
LIN {X 0,Y 601.461,Z 391.121,A -85,B 0,C 180,E1 -838.246,E2 -838.246} C_VEL
LIN {X 0,Y 601.512,Z 381.795,A -85,B 0,C 180,E1 -840.938,E2 -840.938} C_VEL
LIN {X 0,Y 601.586,Z 372.82,A -85,B 0,C 180,E1 -843.63,E2 -843.63} C_VEL
LIN {X 0,Y 601.468,Z 365.753,A -85,B 0,C 180,E1 -845.84,E2 -845.84} C_VEL
LIN {X 0,Y 601.412,Z 365.571,A -85,B 0,C 180,E1 -848.468,E2 -848.468} C_VEL
LIN {X 0,Y 601.413,Z 365.572,A -85,B 0,C 180,E1 -850.876,E2 -850.876} C_VEL
LIN {X 0,Y 601.439,Z 365.568,A -85,B 0,C 180,E1 -853.587,E2 -853.587} C_VEL
LIN {X 0,Y 601.415,Z 365.57,A -85,B 0,C 180,E1 -856.43,E2 -856.43} C_VEL
LIN {X 0,Y 601.42,Z 365.57,A -85,B 0,C 180,E1 -859.126,E2 -859.126} C_VEL
LIN {X 0,Y 601.407,Z 365.571,A -85,B 0,C 180,E1 -861.731,E2 -861.731} C_VEL
LIN {X 0,Y 601.389,Z 365.575,A -85,B 0,C 180,E1 -864.245,E2 -864.245} C_VEL
LIN {X 0,Y 601.425,Z 365.573,A -85,B 0,C 180,E1 -866.686,E2 -866.686} C_VEL
LIN {X 0,Y 601.401,Z 365.574,A -85,B 0,C 180,E1 -869.056,E2 -869.056} C_VEL
LIN {X 0,Y 601.438,Z 365.567,A -85,B 0,C 180,E1 -871.373,E2 -871.373} C_VEL
LIN {X 0,Y 601.408,Z 365.572,A -85,B 0,C 180,E1 -874.381,E2 -874.381} C_VEL
LIN {X 0,Y 601.398,Z 365.572,A -85,B 0,C 180,E1 -876.588,E2 -876.588} C_VEL
LIN {X 0,Y 601.434,Z 365.568,A -85,B 0,C 180,E1 -879.478,E2 -879.478} C_VEL
LIN {X 0,Y 601.392,Z 365.573,A -85,B 0,C 180,E1 -882.311,E2 -882.311} C_VEL
LIN {X 0,Y 601.408,Z 365.572,A -85,B 0,C 180,E1 -884.408,E2 -884.408} C_VEL
LIN {X 0,Y 601.421,Z 365.57,A -85,B 0,C 180,E1 -887.171,E2 -887.171} C_VEL
LIN {X 0,Y 601.4,Z 365.572,A -85,B 0,C 180,E1 -889.904,E2 -889.904} C_VEL
LIN {X 0,Y 601.415,Z 365.57,A -85,B 0,C 180,E1 -892.614,E2 -892.614} C_VEL
LIN {X 0,Y 601.414,Z 365.57,A -85,B 0,C 180,E1 -895.307,E2 -895.307} C_VEL
LIN {X 0,Y 601.406,Z 365.571,A -85,B 0,C 180,E1 -897.99,E2 -897.99} C_VEL
LIN {X 0,Y 601.45,Z 365.566,A -85,B 0,C 180,E1 -900.669,E2 -900.669} C_VEL
LIN {X 0,Y 601.421,Z 365.57,A -85,B 0,C 180,E1 -903.349,E2 -903.349} C_VEL
LIN {X 0,Y 601.394,Z 365.573,A -85,B 0,C 180,E1 -906.037,E2 -906.037} C_VEL
LIN {X 0,Y 601.419,Z 365.57,A -85,B 0,C 180,E1 -908.737,E2 -908.737} C_VEL
LIN {X 0,Y 601.412,Z 365.57,A -85,B 0,C 180,E1 -911.458,E2 -911.458} C_VEL
LIN {X 0,Y 601.405,Z 365.573,A -85,B 0,C 180,E1 -912.355,E2 -912.355} C_VEL
LIN {X 0,Y 600.741,Z 365.654,A -85,B 0,C 180,E1 -912.915,E2 -912.915} C_VEL
LIN {X 0,Y 597.883,Z 366.012,A -85,B 0,C 180,E1 -913.823,E2 -913.823} C_VEL
LIN {X 0,Y 595.467,Z 366.314,A -85,B 0,C 180,E1 -914.553,E2 -914.553} C_VEL
LIN {X 0,Y 594.429,Z 366.443,A -85,B 0,C 180,E1 -915.116,E2 -915.116} C_VEL
LIN {X 0,Y 594.345,Z 366.451,A -85,B 0,C 180,E1 -915.307,E2 -915.307} C_VEL
LIN {X 0,Y 594.391,Z 366.446,A -85,B 0,C 180,E1 -917.193,E2 -917.193} C_VEL
LIN {X 0,Y 594.372,Z 366.449,A -85,B 0,C 180,E1 -920.053,E2 -920.053} C_VEL
LIN {X 0,Y 594.359,Z 366.454,A -85,B 0,C 180,E1 -922.967,E2 -922.967} C_VEL
LIN {X 0,Y 594.38,Z 366.447,A -85,B 0,C 180,E1 -925.192,E2 -925.192} C_VEL
LIN {X 0,Y 594.351,Z 366.45,A -85,B 0,C 180,E1 -927.518,E2 -927.518} C_VEL
LIN {X 0,Y 594.372,Z 366.451,A -85,B 0,C 180,E1 -929.776,E2 -929.776} C_VEL
LIN {X 0,Y 594.371,Z 366.45,A -85,B 0,C 180,E1 -932.146,E2 -932.146} C_VEL
LIN {X 0,Y 594.386,Z 366.446,A -85,B 0,C 180,E1 -934.579,E2 -934.579} C_VEL
LIN {X 0,Y 594.391,Z 366.449,A -85,B 0,C 180,E1 -937.607,E2 -937.607} C_VEL
LIN {X 0,Y 594.364,Z 366.451,A -85,B 0,C 180,E1 -940.566,E2 -940.566} C_VEL
LIN {X 0,Y 594.355,Z 366.451,A -85,B 0,C 180,E1 -943.299,E2 -943.299} C_VEL
LIN {X 0,Y 594.364,Z 366.449,A -85,B 0,C 180,E1 -946.16,E2 -946.16} C_VEL
LIN {X 0,Y 594.37,Z 366.448,A -85,B 0,C 180,E1 -949.177,E2 -949.177} C_VEL
LIN {X 0,Y 594.378,Z 366.449,A -85,B 0,C 180,E1 -951.295,E2 -951.295} C_VEL
LIN {X 0,Y 594.36,Z 366.453,A -85,B 0,C 180,E1 -953.754,E2 -953.754} C_VEL
LIN {X 0,Y 594.379,Z 366.448,A -85,B 0,C 180,E1 -956.237,E2 -956.237} C_VEL
LIN {X 0,Y 594.39,Z 366.445,A -85,B 0,C 180,E1 -958.649,E2 -958.649} C_VEL
LIN {X 0,Y 594.377,Z 366.451,A -85,B 0,C 180,E1 -961.771,E2 -961.771} C_VEL
LIN {X 0,Y 594.379,Z 366.447,A -85,B 0,C 180,E1 -964.054,E2 -964.054} C_VEL
LIN {X 0,Y 594.394,Z 366.445,A -85,B 0,C 180,E1 -966.294,E2 -966.294} C_VEL
LIN {X 0,Y 594.39,Z 366.445,A -85,B 0,C 180,E1 -969.222,E2 -969.222} C_VEL
LIN {X 0,Y 594.354,Z 366.45,A -85,B 0,C 180,E1 -972.093,E2 -972.093} C_VEL
LIN {X 0,Y 594.363,Z 366.45,A -85,B 0,C 180,E1 -974.217,E2 -974.217} C_VEL
LIN {X 0,Y 594.38,Z 366.448,A -85,B 0,C 180,E1 -976.319,E2 -976.319} C_VEL
LIN {X 0,Y 594.377,Z 366.449,A -85,B 0,C 180,E1 -979.093,E2 -979.093} C_VEL
LIN {X 0,Y 594.407,Z 366.446,A -85,B 0,C 180,E1 -981.841,E2 -981.841} C_VEL
LIN {X 0,Y 594.398,Z 366.448,A -85,B 0,C 180,E1 -984.57,E2 -984.57} C_VEL
LIN {X 0,Y 594.407,Z 366.447,A -85,B 0,C 180,E1 -987.287,E2 -987.287} C_VEL
LIN {X 0,Y 594.408,Z 366.448,A -85,B 0,C 180,E1 -989.998,E2 -989.998} C_VEL
LIN {X 0,Y 594.407,Z 366.447,A -85,B 0,C 180,E1 -992.708,E2 -992.708} C_VEL
LIN {X 0,Y 594.398,Z 366.448,A -85,B 0,C 180,E1 -995.425,E2 -995.425} C_VEL
LIN {X 0,Y 594.405,Z 366.447,A -85,B 0,C 180,E1 -998.154,E2 -998.154} C_VEL
LIN {X 0,Y 594.384,Z 366.447,A -85,B 0,C 180,E1 -1001.075,E2 -1001.075} C_VEL
LIN {X 0,Y 594.375,Z 366.449,A -85,B 0,C 180,E1 -1003.676,E2 -1003.676} C_VEL
LIN {X 0,Y 594.378,Z 366.446,A -85,B 0,C 180,E1 -1006.717,E2 -1006.717} C_VEL
LIN {X 0,Y 594.358,Z 366.449,A -85,B 0,C 180,E1 -1009.331,E2 -1009.331} C_VEL
LIN {X 0,Y 594.358,Z 366.454,A -85,B 0,C 180,E1 -1011.5,E2 -1011.5} C_VEL
LIN {X 0,Y 594.371,Z 366.449,A -85,B 0,C 180,E1 -1014.443,E2 -1014.443} C_VEL
LIN {X 0,Y 594.342,Z 366.455,A -85,B 0,C 180,E1 -1016.698,E2 -1016.698} C_VEL
LIN {X 0,Y 594.318,Z 366.727,A -85,B 0,C 180,E1 -1017.516,E2 -1017.516} C_VEL
LIN {X 0,Y 594.271,Z 370.325,A -85,B 0,C 180,E1 -1020.562,E2 -1020.562} C_VEL
LIN {X 0,Y 594.263,Z 373.198,A -85,B 0,C 180,E1 -1022.953,E2 -1022.953} C_VEL
LIN {X 0,Y 594.243,Z 376.151,A -85,B 0,C 180,E1 -1025.412,E2 -1025.412} C_VEL
LIN {X 0,Y 594.228,Z 379.402,A -85,B 0,C 180,E1 -1027.948,E2 -1027.948} C_VEL
LIN {X 0,Y 594.226,Z 382.835,A -85,B 0,C 180,E1 -1030.574,E2 -1030.574} C_VEL
LIN {X 0,Y 594.242,Z 386.473,A -85,B 0,C 180,E1 -1033.306,E2 -1033.306} C_VEL
LIN {X 0,Y 594.217,Z 389.779,A -85,B 0,C 180,E1 -1035.749,E2 -1035.749} C_VEL
LIN {X 0,Y 594.228,Z 393.082,A -85,B 0,C 180,E1 -1038.163,E2 -1038.163} C_VEL
LIN {X 0,Y 594.228,Z 395.685,A -85,B 0,C 180,E1 -1040.046,E2 -1040.046} C_VEL
LIN {X 0,Y 594.657,Z 401.147,A -85,B 0,C 180,E1 -1040.167,E2 -1040.167} C_VEL
LIN {X 0,Y 594.594,Z 413.366,A -85,B 0,C 180,E1 -1040.503,E2 -1040.503} C_VEL
LIN {X 0,Y 594.541,Z 425.946,A -85,B 0,C 180,E1 -1040.991,E2 -1040.991} C_VEL
LIN {X 0,Y 594.498,Z 436.565,A -85,B 0,C 180,E1 -1041.53,E2 -1041.53} C_VEL
LIN {X 0,Y 594.457,Z 447.832,A -85,B 0,C 180,E1 -1042.253,E2 -1042.253} C_VEL
LIN {X 0,Y 594.411,Z 458.137,A -85,B 0,C 180,E1 -1043.079,E2 -1043.079} C_VEL
LIN {X 0,Y 594.379,Z 467.176,A -85,B 0,C 180,E1 -1043.968,E2 -1043.968} C_VEL
LIN {X 0,Y 594.306,Z 474.61,A -85,B 0,C 180,E1 -1044.859,E2 -1044.859} C_VEL
LIN {X 0,Y 594.293,Z 481.461,A -85,B 0,C 180,E1 -1045.867,E2 -1045.867} C_VEL
LIN {X 0,Y 594.271,Z 487.781,A -85,B 0,C 180,E1 -1047.044,E2 -1047.044} C_VEL
LIN {X 0,Y 594.248,Z 491.206,A -85,B 0,C 180,E1 -1047.847,E2 -1047.847} C_VEL
LIN {X 0,Y 594.245,Z 495.044,A -85,B 0,C 180,E1 -1049.039,E2 -1049.039} C_VEL
LIN {X 0,Y 594.232,Z 497.535,A -85,B 0,C 180,E1 -1050.217,E2 -1050.217} C_VEL
LIN {X 0,Y 594.233,Z 498.572,A -85,B 0,C 180,E1 -1051.06,E2 -1051.06} C_VEL
LIN {X 0,Y 594.217,Z 498.942,A -85,B 0,C 180,E1 -1051.766,E2 -1051.766} C_VEL
LIN {X 0,Y 594.234,Z 498.894,A -85,B 0,C 180,E1 -1052.533,E2 -1052.533} C_VEL
LIN {X 0,Y 594.215,Z 498.308,A -85,B 0,C 180,E1 -1053.293,E2 -1053.293} C_VEL
LIN {X 0,Y 594.234,Z 497.248,A -85,B 0,C 180,E1 -1054.05,E2 -1054.05} C_VEL
LIN {X 0,Y 594.254,Z 494.716,A -85,B 0,C 180,E1 -1055.176,E2 -1055.176} C_VEL
LIN {X 0,Y 594.27,Z 491.028,A -85,B 0,C 180,E1 -1056.292,E2 -1056.292} C_VEL
LIN {X 0,Y 594.269,Z 485.452,A -85,B 0,C 180,E1 -1057.517,E2 -1057.517} C_VEL
LIN {X 0,Y 594.324,Z 478.636,A -85,B 0,C 180,E1 -1058.663,E2 -1058.663} C_VEL
LIN {X 0,Y 594.334,Z 471.81,A -85,B 0,C 180,E1 -1059.585,E2 -1059.585} C_VEL
LIN {X 0,Y 594.362,Z 463.706,A -85,B 0,C 180,E1 -1060.487,E2 -1060.487} C_VEL
LIN {X 0,Y 594.436,Z 453.732,A -85,B 0,C 180,E1 -1061.385,E2 -1061.385} C_VEL
LIN {X 0,Y 594.435,Z 442.72,A -85,B 0,C 180,E1 -1062.187,E2 -1062.187} C_VEL
LIN {X 0,Y 594.48,Z 431.98,A -85,B 0,C 180,E1 -1062.81,E2 -1062.81} C_VEL
LIN {X 0,Y 594.569,Z 420.384,A -85,B 0,C 180,E1 -1063.334,E2 -1063.334} C_VEL
LIN {X 0,Y 594.634,Z 407.489,A -85,B 0,C 180,E1 -1063.765,E2 -1063.765} C_VEL
LIN {X 0,Y 594.459,Z 397.482,A -85,B 0,C 180,E1 -1064.002,E2 -1064.002} C_VEL
LIN {X 0,Y 594.238,Z 395.66,A -85,B 0,C 180,E1 -1064.062,E2 -1064.062} C_VEL
LIN {X 0,Y 594.211,Z 391.59,A -85,B 0,C 180,E1 -1067.014,E2 -1067.014} C_VEL
LIN {X 0,Y 594.182,Z 387.826,A -85,B 0,C 180,E1 -1069.781,E2 -1069.781} C_VEL
LIN {X 0,Y 594.221,Z 384.148,A -85,B 0,C 180,E1 -1072.525,E2 -1072.525} C_VEL
LIN {X 0,Y 594.254,Z 380.557,A -85,B 0,C 180,E1 -1075.252,E2 -1075.252} C_VEL
LIN {X 0,Y 594.202,Z 377.058,A -85,B 0,C 180,E1 -1077.967,E2 -1077.967} C_VEL
LIN {X 0,Y 594.313,Z 373.823,A -85,B 0,C 180,E1 -1080.678,E2 -1080.678} C_VEL
LIN {X 0,Y 594.293,Z 370.697,A -85,B 0,C 180,E1 -1083.39,E2 -1083.39} C_VEL
LIN {X 0,Y 594.326,Z 367.507,A -85,B 0,C 180,E1 -1086.11,E2 -1086.11} C_VEL
LIN {X 0,Y 594.321,Z 366.702,A -85,B 0,C 180,E1 -1086.792,E2 -1086.792} C_VEL
LIN {X 0,Y 594.374,Z 366.452,A -85,B 0,C 180,E1 -1088.843,E2 -1088.843} C_VEL
LIN {X 0,Y 594.371,Z 366.45,A -85,B 0,C 180,E1 -1091.597,E2 -1091.597} C_VEL
LIN {X 0,Y 594.354,Z 366.45,A -85,B 0,C 180,E1 -1094.378,E2 -1094.378} C_VEL
LIN {X 0,Y 594.372,Z 366.447,A -85,B 0,C 180,E1 -1097.194,E2 -1097.194} C_VEL
LIN {X 0,Y 594.349,Z 366.453,A -85,B 0,C 180,E1 -1099.336,E2 -1099.336} C_VEL
LIN {X 0,Y 594.349,Z 366.449,A -85,B 0,C 180,E1 -1101.504,E2 -1101.504} C_VEL
LIN {X 0,Y 594.378,Z 366.451,A -85,B 0,C 180,E1 -1103.705,E2 -1103.705} C_VEL
LIN {X 0,Y 594.361,Z 366.452,A -85,B 0,C 180,E1 -1106.701,E2 -1106.701} C_VEL
LIN {X 0,Y 594.394,Z 366.444,A -85,B 0,C 180,E1 -1108.998,E2 -1108.998} C_VEL
LIN {X 0,Y 594.366,Z 366.447,A -85,B 0,C 180,E1 -1111.648,E2 -1111.648} C_VEL
LIN {X 0,Y 594.382,Z 366.445,A -85,B 0,C 180,E1 -1114.58,E2 -1114.58} C_VEL
LIN {X 0,Y 594.367,Z 366.452,A -85,B 0,C 180,E1 -1117.089,E2 -1117.089} C_VEL
LIN {X 0,Y 594.372,Z 366.45,A -85,B 0,C 180,E1 -1119.78,E2 -1119.78} C_VEL
LIN {X 0,Y 594.37,Z 366.447,A -85,B 0,C 180,E1 -1122.376,E2 -1122.376} C_VEL
LIN {X 0,Y 594.339,Z 366.451,A -85,B 0,C 180,E1 -1125.194,E2 -1125.194} C_VEL
LIN {X 0,Y 594.37,Z 366.45,A -85,B 0,C 180,E1 -1127.63,E2 -1127.63} C_VEL
LIN {X 0,Y 594.374,Z 366.453,A -85,B 0,C 180,E1 -1130.324,E2 -1130.324} C_VEL
LIN {X 0,Y 594.374,Z 366.45,A -85,B 0,C 180,E1 -1132.917,E2 -1132.917} C_VEL
LIN {X 0,Y 594.386,Z 366.515,A -85,B 0,C 180,E1 -1133.867,E2 -1133.867} C_VEL
LIN {X 0,Y 594.626,Z 371.26,A -85,B 0,C 180,E1 -1135.441,E2 -1135.441} C_VEL
LIN {X 0,Y 594.539,Z 379.016,A -85,B 0,C 180,E1 -1137.867,E2 -1137.867} C_VEL
LIN {X 0,Y 594.497,Z 388.453,A -85,B 0,C 180,E1 -1140.624,E2 -1140.624} C_VEL
LIN {X 0,Y 594.429,Z 396.436,A -85,B 0,C 180,E1 -1142.927,E2 -1142.927} C_VEL
LIN {X 0,Y 594.443,Z 404.379,A -85,B 0,C 180,E1 -1145.187,E2 -1145.187} C_VEL
LIN {X 0,Y 594.413,Z 413.646,A -85,B 0,C 180,E1 -1147.772,E2 -1147.772} C_VEL
LIN {X 0,Y 594.376,Z 424.237,A -85,B 0,C 180,E1 -1150.669,E2 -1150.669} C_VEL
LIN {X 0,Y 594.313,Z 434.828,A -85,B 0,C 180,E1 -1153.515,E2 -1153.515} C_VEL
LIN {X 0,Y 594.31,Z 445.419,A -85,B 0,C 180,E1 -1156.322,E2 -1156.322} C_VEL
LIN {X 0,Y 594.313,Z 451.746,A -85,B 0,C 180,E1 -1157.943,E2 -1157.943} C_VEL
LIN {X 0,Y 594.675,Z 457.384,A -85,B 0,C 180,E1 -1158.045,E2 -1158.045} C_VEL
LIN {X 0,Y 594.621,Z 470.599,A -85,B 0,C 180,E1 -1158.368,E2 -1158.368} C_VEL
LIN {X 0,Y 594.534,Z 482.605,A -85,B 0,C 180,E1 -1158.799,E2 -1158.799} C_VEL
LIN {X 0,Y 594.482,Z 494.261,A -85,B 0,C 180,E1 -1159.358,E2 -1159.358} C_VEL
LIN {X 0,Y 594.47,Z 505.519,A -85,B 0,C 180,E1 -1160.046,E2 -1160.046} C_VEL
LIN {X 0,Y 594.405,Z 515.68,A -85,B 0,C 180,E1 -1160.818,E2 -1160.818} C_VEL
LIN {X 0,Y 594.371,Z 524.814,A -85,B 0,C 180,E1 -1161.674,E2 -1161.674} C_VEL
LIN {X 0,Y 594.315,Z 533.713,A -85,B 0,C 180,E1 -1162.699,E2 -1162.699} C_VEL
LIN {X 0,Y 594.281,Z 540.175,A -85,B 0,C 180,E1 -1163.616,E2 -1163.616} C_VEL
LIN {X 0,Y 594.289,Z 545.695,A -85,B 0,C 180,E1 -1164.574,E2 -1164.574} C_VEL
LIN {X 0,Y 594.27,Z 550.382,A -85,B 0,C 180,E1 -1165.594,E2 -1165.594} C_VEL
LIN {X 0,Y 594.267,Z 553.964,A -85,B 0,C 180,E1 -1166.613,E2 -1166.613} C_VEL
LIN {X 0,Y 594.225,Z 555.815,A -85,B 0,C 180,E1 -1167.291,E2 -1167.291} C_VEL
LIN {X 0,Y 594.242,Z 557.206,A -85,B 0,C 180,E1 -1167.969,E2 -1167.969} C_VEL
LIN {X 0,Y 594.239,Z 558.786,A -85,B 0,C 180,E1 -1169.325,E2 -1169.325} C_VEL
LIN {X 0,Y 594.236,Z 559,A -85,B 0,C 180,E1 -1170.002,E2 -1170.002} C_VEL
LIN {X 0,Y 594.247,Z 558.182,A -85,B 0,C 180,E1 -1171.358,E2 -1171.358} C_VEL
LIN {X 0,Y 594.242,Z 557.198,A -85,B 0,C 180,E1 -1172.036,E2 -1172.036} C_VEL
LIN {X 0,Y 594.226,Z 555.804,A -85,B 0,C 180,E1 -1172.714,E2 -1172.714} C_VEL
LIN {X 0,Y 594.289,Z 552.888,A -85,B 0,C 180,E1 -1173.732,E2 -1173.732} C_VEL
LIN {X 0,Y 594.241,Z 548.94,A -85,B 0,C 180,E1 -1174.751,E2 -1174.751} C_VEL
LIN {X 0,Y 594.304,Z 542.864,A -85,B 0,C 180,E1 -1175.942,E2 -1175.942} C_VEL
LIN {X 0,Y 594.31,Z 536.219,A -85,B 0,C 180,E1 -1176.964,E2 -1176.964} C_VEL
LIN {X 0,Y 594.36,Z 527.97,A -85,B 0,C 180,E1 -1177.989,E2 -1177.989} C_VEL
LIN {X 0,Y 594.383,Z 519.512,A -85,B 0,C 180,E1 -1178.844,E2 -1178.844} C_VEL
LIN {X 0,Y 594.435,Z 509.064,A -85,B 0,C 180,E1 -1179.702,E2 -1179.702} C_VEL
LIN {X 0,Y 594.464,Z 498.723,A -85,B 0,C 180,E1 -1180.389,E2 -1180.389} C_VEL
LIN {X 0,Y 594.506,Z 486.723,A -85,B 0,C 180,E1 -1181.021,E2 -1181.021} C_VEL
LIN {X 0,Y 594.567,Z 474.426,A -85,B 0,C 180,E1 -1181.507,E2 -1181.507} C_VEL
LIN {X 0,Y 594.655,Z 461.346,A -85,B 0,C 180,E1 -1181.874,E2 -1181.874} C_VEL
LIN {X 0,Y 594.46,Z 452.9,A -85,B 0,C 180,E1 -1182.037,E2 -1182.037} C_VEL
LIN {X 0,Y 594.296,Z 451.522,A -85,B 0,C 180,E1 -1182.076,E2 -1182.076} C_VEL
LIN {X 0,Y 594.315,Z 441.428,A -85,B 0,C 180,E1 -1184.731,E2 -1184.731} C_VEL
LIN {X 0,Y 594.336,Z 430.837,A -85,B 0,C 180,E1 -1187.552,E2 -1187.552} C_VEL
LIN {X 0,Y 594.393,Z 421.57,A -85,B 0,C 180,E1 -1190.055,E2 -1190.055} C_VEL
LIN {X 0,Y 594.403,Z 410.979,A -85,B 0,C 180,E1 -1192.968,E2 -1192.968} C_VEL
LIN {X 0,Y 594.465,Z 401.712,A -85,B 0,C 180,E1 -1195.566,E2 -1195.566} C_VEL
LIN {X 0,Y 594.491,Z 392.445,A -85,B 0,C 180,E1 -1198.223,E2 -1198.223} C_VEL
LIN {X 0,Y 594.523,Z 383.045,A -85,B 0,C 180,E1 -1200.947,E2 -1200.947} C_VEL
LIN {X 0,Y 594.632,Z 373.877,A -85,B 0,C 180,E1 -1203.747,E2 -1203.747} C_VEL
LIN {X 0,Y 594.55,Z 367.357,A -85,B 0,C 180,E1 -1205.813,E2 -1205.813} C_VEL
LIN {X 0,Y 594.379,Z 366.45,A -85,B 0,C 180,E1 -1206.139,E2 -1206.139} C_VEL
LIN {X 0,Y 594.375,Z 366.448,A -85,B 0,C 180,E1 -1208.807,E2 -1208.807} C_VEL
LIN {X 0,Y 594.383,Z 366.451,A -85,B 0,C 180,E1 -1211.848,E2 -1211.848} C_VEL
LIN {X 0,Y 594.371,Z 366.449,A -85,B 0,C 180,E1 -1214.239,E2 -1214.239} C_VEL
LIN {X 0,Y 594.347,Z 366.454,A -85,B 0,C 180,E1 -1217.151,E2 -1217.151} C_VEL
LIN {X 0,Y 594.379,Z 366.447,A -85,B 0,C 180,E1 -1219.433,E2 -1219.433} C_VEL
LIN {X 0,Y 594.394,Z 366.447,A -85,B 0,C 180,E1 -1222.393,E2 -1222.393} C_VEL
LIN {X 0,Y 594.381,Z 366.449,A -85,B 0,C 180,E1 -1225.42,E2 -1225.42} C_VEL
LIN {X 0,Y 594.38,Z 366.447,A -85,B 0,C 180,E1 -1228.359,E2 -1228.359} C_VEL
LIN {X 0,Y 594.392,Z 366.446,A -85,B 0,C 180,E1 -1231.043,E2 -1231.043} C_VEL
LIN {X 0,Y 594.366,Z 366.448,A -85,B 0,C 180,E1 -1234.055,E2 -1234.055} C_VEL
LIN {X 0,Y 594.381,Z 366.448,A -85,B 0,C 180,E1 -1236.295,E2 -1236.295} C_VEL
LIN {X 0,Y 594.41,Z 366.443,A -85,B 0,C 180,E1 -1239.224,E2 -1239.224} C_VEL
LIN {X 0,Y 594.346,Z 366.45,A -85,B 0,C 180,E1 -1242.094,E2 -1242.094} C_VEL
LIN {X 0,Y 594.364,Z 366.451,A -85,B 0,C 180,E1 -1244.218,E2 -1244.218} C_VEL
LIN {X 0,Y 594.369,Z 366.448,A -85,B 0,C 180,E1 -1246.32,E2 -1246.32} C_VEL
LIN {X 0,Y 594.382,Z 366.447,A -85,B 0,C 180,E1 -1249.094,E2 -1249.094} C_VEL
LIN {X 0,Y 594.387,Z 366.447,A -85,B 0,C 180,E1 -1251.842,E2 -1251.842} C_VEL
LIN {X 0,Y 594.391,Z 366.447,A -85,B 0,C 180,E1 -1254.572,E2 -1254.572} C_VEL
LIN {X 0,Y 594.417,Z 366.444,A -85,B 0,C 180,E1 -1257.289,E2 -1257.289} C_VEL
LIN {X 0,Y 594.416,Z 366.445,A -85,B 0,C 180,E1 -1259.999,E2 -1259.999} C_VEL
LIN {X 0,Y 594.401,Z 366.447,A -85,B 0,C 180,E1 -1262.71,E2 -1262.71} C_VEL
LIN {X 0,Y 594.393,Z 366.449,A -85,B 0,C 180,E1 -1265.427,E2 -1265.427} C_VEL
LIN {X 0,Y 594.367,Z 366.452,A -85,B 0,C 180,E1 -1268.157,E2 -1268.157} C_VEL
LIN {X 0,Y 594.389,Z 366.448,A -85,B 0,C 180,E1 -1271.069,E2 -1271.069} C_VEL
LIN {X 0,Y 594.371,Z 366.451,A -85,B 0,C 180,E1 -1273.678,E2 -1273.678} C_VEL
LIN {X 0,Y 594.345,Z 366.451,A -85,B 0,C 180,E1 -1275.307,E2 -1275.307} C_VEL
LIN {X 0,Y 593.676,Z 366.536,A -85,B 0,C 180,E1 -1275.873,E2 -1275.873} C_VEL
LIN {X 0,Y 590.811,Z 366.891,A -85,B 0,C 180,E1 -1276.791,E2 -1276.791} C_VEL
LIN {X 0,Y 588.4,Z 367.195,A -85,B 0,C 180,E1 -1277.53,E2 -1277.53} C_VEL
LIN {X 0,Y 587.379,Z 367.319,A -85,B 0,C 180,E1 -1278.1,E2 -1278.1} C_VEL
LIN {X 0,Y 587.303,Z 367.328,A -85,B 0,C 180,E1 -1278.293,E2 -1278.293} C_VEL
LIN {X 0,Y 587.337,Z 367.324,A -85,B 0,C 180,E1 -1281.037,E2 -1281.037} C_VEL
LIN {X 0,Y 587.315,Z 367.328,A -85,B 0,C 180,E1 -1283.258,E2 -1283.258} C_VEL
LIN {X 0,Y 587.339,Z 367.327,A -85,B 0,C 180,E1 -1285.516,E2 -1285.516} C_VEL
LIN {X 0,Y 587.311,Z 367.327,A -85,B 0,C 180,E1 -1287.819,E2 -1287.819} C_VEL
LIN {X 0,Y 587.327,Z 367.325,A -85,B 0,C 180,E1 -1290.506,E2 -1290.506} C_VEL
LIN {X 0,Y 587.338,Z 367.325,A -85,B 0,C 180,E1 -1293.396,E2 -1293.396} C_VEL
LIN {X 0,Y 587.292,Z 367.329,A -85,B 0,C 180,E1 -1295.899,E2 -1295.899} C_VEL
LIN {X 0,Y 587.332,Z 367.324,A -85,B 0,C 180,E1 -1298.478,E2 -1298.478} C_VEL
LIN {X 0,Y 587.334,Z 367.324,A -85,B 0,C 180,E1 -1301.156,E2 -1301.156} C_VEL
LIN {X 0,Y 587.306,Z 367.329,A -85,B 0,C 180,E1 -1304.109,E2 -1304.109} C_VEL
LIN {X 0,Y 587.303,Z 367.332,A -85,B 0,C 180,E1 -1306.991,E2 -1306.991} C_VEL
LIN {X 0,Y 587.317,Z 367.33,A -85,B 0,C 180,E1 -1309.744,E2 -1309.744} C_VEL
LIN {X 0,Y 587.34,Z 367.327,A -85,B 0,C 180,E1 -1312.39,E2 -1312.39} C_VEL
LIN {X 0,Y 587.351,Z 367.325,A -85,B 0,C 180,E1 -1314.944,E2 -1314.944} C_VEL
LIN {X 0,Y 587.338,Z 367.324,A -85,B 0,C 180,E1 -1317.419,E2 -1317.419} C_VEL
LIN {X 0,Y 587.317,Z 367.326,A -85,B 0,C 180,E1 -1319.827,E2 -1319.827} C_VEL
LIN {X 0,Y 587.352,Z 367.322,A -85,B 0,C 180,E1 -1322.305,E2 -1322.305} C_VEL
LIN {X 0,Y 587.336,Z 367.328,A -85,B 0,C 180,E1 -1324.482,E2 -1324.482} C_VEL
LIN {X 0,Y 587.32,Z 367.33,A -85,B 0,C 180,E1 -1327.129,E2 -1327.129} C_VEL
LIN {X 0,Y 587.321,Z 367.328,A -85,B 0,C 180,E1 -1329.693,E2 -1329.693} C_VEL
LIN {X 0,Y 587.309,Z 367.327,A -85,B 0,C 180,E1 -1331.871,E2 -1331.871} C_VEL
LIN {X 0,Y 587.317,Z 367.33,A -85,B 0,C 180,E1 -1334.023,E2 -1334.023} C_VEL
LIN {X 0,Y 587.358,Z 367.322,A -85,B 0,C 180,E1 -1336.152,E2 -1336.152} C_VEL
LIN {X 0,Y 587.341,Z 367.325,A -85,B 0,C 180,E1 -1338.96,E2 -1338.96} C_VEL
LIN {X 0,Y 587.359,Z 367.323,A -85,B 0,C 180,E1 -1341.742,E2 -1341.742} C_VEL
LIN {X 0,Y 587.365,Z 367.324,A -85,B 0,C 180,E1 -1344.505,E2 -1344.505} C_VEL
LIN {X 0,Y 587.374,Z 367.319,A -85,B 0,C 180,E1 -1347.94,E2 -1347.94} C_VEL
LIN {X 0,Y 587.373,Z 367.319,A -85,B 0,C 180,E1 -1350.683,E2 -1350.683} C_VEL
LIN {X 0,Y 587.315,Z 367.326,A -85,B 0,C 180,E1 -1353.428,E2 -1353.428} C_VEL
LIN {X 0,Y 587.342,Z 367.323,A -85,B 0,C 180,E1 -1356.18,E2 -1356.18} C_VEL
LIN {X 0,Y 587.317,Z 367.327,A -85,B 0,C 180,E1 -1358.947,E2 -1358.947} C_VEL
LIN {X 0,Y 587.331,Z 367.326,A -85,B 0,C 180,E1 -1361.734,E2 -1361.734} C_VEL
LIN {X 0,Y 587.327,Z 367.328,A -85,B 0,C 180,E1 -1364.551,E2 -1364.551} C_VEL
LIN {X 0,Y 587.347,Z 367.327,A -85,B 0,C 180,E1 -1367.403,E2 -1367.403} C_VEL
LIN {X 0,Y 587.316,Z 367.329,A -85,B 0,C 180,E1 -1370.302,E2 -1370.302} C_VEL
LIN {X 0,Y 587.345,Z 367.323,A -85,B 0,C 180,E1 -1373.254,E2 -1373.254} C_VEL
LIN {X 0,Y 587.341,Z 367.323,A -85,B 0,C 180,E1 -1376.275,E2 -1376.275} C_VEL
LIN {X 0,Y 587.242,Z 367.694,A -85,B 0,C 180,E1 -1377.819,E2 -1377.819} C_VEL
LIN {X 0,Y 587.229,Z 370.826,A -85,B 0,C 180,E1 -1380.494,E2 -1380.494} C_VEL
LIN {X 0,Y 587.177,Z 374.286,A -85,B 0,C 180,E1 -1383.403,E2 -1383.403} C_VEL
LIN {X 0,Y 587.162,Z 377.204,A -85,B 0,C 180,E1 -1385.905,E2 -1385.905} C_VEL
LIN {X 0,Y 587.144,Z 381.046,A -85,B 0,C 180,E1 -1388.92,E2 -1388.92} C_VEL
LIN {X 0,Y 587.14,Z 383.967,A -85,B 0,C 180,E1 -1391.169,E2 -1391.169} C_VEL
LIN {X 0,Y 587.15,Z 387.656,A -85,B 0,C 180,E1 -1393.962,E2 -1393.962} C_VEL
LIN {X 0,Y 587.15,Z 390.433,A -85,B 0,C 180,E1 -1396.034,E2 -1396.034} C_VEL
LIN {X 0,Y 587.104,Z 394.218,A -85,B 0,C 180,E1 -1398.824,E2 -1398.824} C_VEL
LIN {X 0,Y 587.147,Z 395.67,A -85,B 0,C 180,E1 -1399.888,E2 -1399.888} C_VEL
LIN {X 0,Y 587.731,Z 401.258,A -85,B 0,C 180,E1 -1400.027,E2 -1400.027} C_VEL
LIN {X 0,Y 587.627,Z 414.038,A -85,B 0,C 180,E1 -1400.387,E2 -1400.387} C_VEL
LIN {X 0,Y 587.563,Z 426.853,A -85,B 0,C 180,E1 -1400.898,E2 -1400.898} C_VEL
LIN {X 0,Y 587.473,Z 438.75,A -85,B 0,C 180,E1 -1401.533,E2 -1401.533} C_VEL
LIN {X 0,Y 587.416,Z 449.667,A -85,B 0,C 180,E1 -1402.271,E2 -1402.271} C_VEL
LIN {X 0,Y 587.347,Z 460.078,A -85,B 0,C 180,E1 -1403.147,E2 -1403.147} C_VEL
LIN {X 0,Y 587.278,Z 469.179,A -85,B 0,C 180,E1 -1404.1,E2 -1404.1} C_VEL
LIN {X 0,Y 587.24,Z 477.208,A -85,B 0,C 180,E1 -1405.135,E2 -1405.135} C_VEL
LIN {X 0,Y 587.212,Z 483.75,A -85,B 0,C 180,E1 -1406.185,E2 -1406.185} C_VEL
LIN {X 0,Y 587.157,Z 489.66,A -85,B 0,C 180,E1 -1407.411,E2 -1407.411} C_VEL
LIN {X 0,Y 587.168,Z 493.988,A -85,B 0,C 180,E1 -1408.624,E2 -1408.624} C_VEL
LIN {X 0,Y 587.154,Z 496.909,A -85,B 0,C 180,E1 -1409.821,E2 -1409.821} C_VEL
LIN {X 0,Y 587.142,Z 498.436,A -85,B 0,C 180,E1 -1410.895,E2 -1410.895} C_VEL
LIN {X 0,Y 587.132,Z 498.94,A -85,B 0,C 180,E1 -1412.339,E2 -1412.339} C_VEL
LIN {X 0,Y 587.139,Z 497.827,A -85,B 0,C 180,E1 -1413.713,E2 -1413.713} C_VEL
LIN {X 0,Y 587.124,Z 496.481,A -85,B 0,C 180,E1 -1414.474,E2 -1414.474} C_VEL
LIN {X 0,Y 587.163,Z 494.036,A -85,B 0,C 180,E1 -1415.45,E2 -1415.45} C_VEL
LIN {X 0,Y 587.187,Z 489.424,A -85,B 0,C 180,E1 -1416.736,E2 -1416.736} C_VEL
LIN {X 0,Y 587.22,Z 484.03,A -85,B 0,C 180,E1 -1417.853,E2 -1417.853} C_VEL
LIN {X 0,Y 587.255,Z 477.1,A -85,B 0,C 180,E1 -1418.97,E2 -1418.97} C_VEL
LIN {X 0,Y 587.291,Z 468.579,A -85,B 0,C 180,E1 -1420.06,E2 -1420.06} C_VEL
LIN {X 0,Y 587.349,Z 460.05,A -85,B 0,C 180,E1 -1420.946,E2 -1420.946} C_VEL
LIN {X 0,Y 587.404,Z 450.099,A -85,B 0,C 180,E1 -1421.786,E2 -1421.786} C_VEL
LIN {X 0,Y 587.459,Z 439.548,A -85,B 0,C 180,E1 -1422.508,E2 -1422.508} C_VEL
LIN {X 0,Y 587.536,Z 428.525,A -85,B 0,C 180,E1 -1423.111,E2 -1423.111} C_VEL
LIN {X 0,Y 587.617,Z 416.143,A -85,B 0,C 180,E1 -1423.632,E2 -1423.632} C_VEL
LIN {X 0,Y 587.682,Z 403.369,A -85,B 0,C 180,E1 -1424.013,E2 -1424.013} C_VEL
LIN {X 0,Y 587.44,Z 397.851,A -85,B 0,C 180,E1 -1424.14,E2 -1424.14} C_VEL
LIN {X 0,Y 587.13,Z 395.676,A -85,B 0,C 180,E1 -1424.198,E2 -1424.198} C_VEL
LIN {X 0,Y 587.106,Z 392.058,A -85,B 0,C 180,E1 -1426.854,E2 -1426.854} C_VEL
LIN {X 0,Y 587.097,Z 388.288,A -85,B 0,C 180,E1 -1429.656,E2 -1429.656} C_VEL
LIN {X 0,Y 587.135,Z 384.606,A -85,B 0,C 180,E1 -1432.435,E2 -1432.435} C_VEL
LIN {X 0,Y 587.159,Z 381.013,A -85,B 0,C 180,E1 -1435.194,E2 -1435.194} C_VEL
LIN {X 0,Y 587.114,Z 377.512,A -85,B 0,C 180,E1 -1437.943,E2 -1437.943} C_VEL
LIN {X 0,Y 587.26,Z 374.561,A -85,B 0,C 180,E1 -1440.686,E2 -1440.686} C_VEL
LIN {X 0,Y 587.223,Z 371.305,A -85,B 0,C 180,E1 -1443.431,E2 -1443.431} C_VEL
LIN {X 0,Y 587.27,Z 368.075,A -85,B 0,C 180,E1 -1446.184,E2 -1446.184} C_VEL
LIN {X 0,Y 587.275,Z 367.336,A -85,B 0,C 180,E1 -1446.874,E2 -1446.874} C_VEL
LIN {X 0,Y 587.32,Z 367.329,A -85,B 0,C 180,E1 -1448.95,E2 -1448.95} C_VEL
LIN {X 0,Y 587.321,Z 367.33,A -85,B 0,C 180,E1 -1451.738,E2 -1451.738} C_VEL
LIN {X 0,Y 587.305,Z 367.33,A -85,B 0,C 180,E1 -1454.555,E2 -1454.555} C_VEL
LIN {X 0,Y 587.338,Z 367.324,A -85,B 0,C 180,E1 -1457.407,E2 -1457.407} C_VEL
LIN {X 0,Y 587.321,Z 367.326,A -85,B 0,C 180,E1 -1459.576,E2 -1459.576} C_VEL
LIN {X 0,Y 587.345,Z 367.323,A -85,B 0,C 180,E1 -1462.514,E2 -1462.514} C_VEL
LIN {X 0,Y 587.31,Z 367.327,A -85,B 0,C 180,E1 -1465.518,E2 -1465.518} C_VEL
LIN {X 0,Y 587.321,Z 367.327,A -85,B 0,C 180,E1 -1467.82,E2 -1467.82} C_VEL
LIN {X 0,Y 587.325,Z 367.325,A -85,B 0,C 180,E1 -1470.516,E2 -1470.516} C_VEL
LIN {X 0,Y 587.311,Z 367.326,A -85,B 0,C 180,E1 -1473.399,E2 -1473.399} C_VEL
LIN {X 0,Y 587.336,Z 367.324,A -85,B 0,C 180,E1 -1475.897,E2 -1475.897} C_VEL
LIN {X 0,Y 587.307,Z 367.332,A -85,B 0,C 180,E1 -1478.482,E2 -1478.482} C_VEL
LIN {X 0,Y 587.343,Z 367.325,A -85,B 0,C 180,E1 -1481.157,E2 -1481.157} C_VEL
LIN {X 0,Y 587.31,Z 367.329,A -85,B 0,C 180,E1 -1484.117,E2 -1484.117} C_VEL
LIN {X 0,Y 587.317,Z 367.327,A -85,B 0,C 180,E1 -1486.999,E2 -1486.999} C_VEL
LIN {X 0,Y 587.298,Z 367.329,A -85,B 0,C 180,E1 -1489.749,E2 -1489.749} C_VEL
LIN {X 0,Y 587.333,Z 367.326,A -85,B 0,C 180,E1 -1492.396,E2 -1492.396} C_VEL
LIN {X 0,Y 587.364,Z 367.52,A -85,B 0,C 180,E1 -1493.685,E2 -1493.685} C_VEL
LIN {X 0,Y 587.671,Z 371.244,A -85,B 0,C 180,E1 -1494.972,E2 -1494.972} C_VEL
LIN {X 0,Y 587.607,Z 378.974,A -85,B 0,C 180,E1 -1497.442,E2 -1497.442} C_VEL
LIN {X 0,Y 587.536,Z 388.334,A -85,B 0,C 180,E1 -1500.241,E2 -1500.241} C_VEL
LIN {X 0,Y 587.421,Z 397.76,A -85,B 0,C 180,E1 -1502.962,E2 -1502.962} C_VEL
LIN {X 0,Y 587.433,Z 405.703,A -85,B 0,C 180,E1 -1505.249,E2 -1505.249} C_VEL
LIN {X 0,Y 587.399,Z 414.97,A -85,B 0,C 180,E1 -1507.863,E2 -1507.863} C_VEL
LIN {X 0,Y 587.32,Z 424.237,A -85,B 0,C 180,E1 -1510.428,E2 -1510.428} C_VEL
LIN {X 0,Y 587.279,Z 434.828,A -85,B 0,C 180,E1 -1513.312,E2 -1513.312} C_VEL
LIN {X 0,Y 587.239,Z 445.419,A -85,B 0,C 180,E1 -1516.154,E2 -1516.154} C_VEL
LIN {X 0,Y 587.219,Z 451.65,A -85,B 0,C 180,E1 -1517.794,E2 -1517.794} C_VEL
LIN {X 0,Y 587.729,Z 457.384,A -85,B 0,C 180,E1 -1517.902,E2 -1517.902} C_VEL
LIN {X 0,Y 587.689,Z 470.599,A -85,B 0,C 180,E1 -1518.229,E2 -1518.229} C_VEL
LIN {X 0,Y 587.566,Z 482.39,A -85,B 0,C 180,E1 -1518.655,E2 -1518.655} C_VEL
LIN {X 0,Y 587.481,Z 494.263,A -85,B 0,C 180,E1 -1519.23,E2 -1519.23} C_VEL
LIN {X 0,Y 587.467,Z 505.521,A -85,B 0,C 180,E1 -1519.926,E2 -1519.926} C_VEL
LIN {X 0,Y 587.383,Z 515.68,A -85,B 0,C 180,E1 -1520.707,E2 -1520.707} C_VEL
LIN {X 0,Y 587.338,Z 524.814,A -85,B 0,C 180,E1 -1521.574,E2 -1521.574} C_VEL
LIN {X 0,Y 587.257,Z 533.712,A -85,B 0,C 180,E1 -1522.611,E2 -1522.611} C_VEL
LIN {X 0,Y 587.195,Z 540.751,A -85,B 0,C 180,E1 -1523.628,E2 -1523.628} C_VEL
LIN {X 0,Y 587.211,Z 545.694,A -85,B 0,C 180,E1 -1524.508,E2 -1524.508} C_VEL
LIN {X 0,Y 587.188,Z 550.382,A -85,B 0,C 180,E1 -1525.541,E2 -1525.541} C_VEL
LIN {X 0,Y 587.193,Z 553.965,A -85,B 0,C 180,E1 -1526.572,E2 -1526.572} C_VEL
LIN {X 0,Y 587.132,Z 555.815,A -85,B 0,C 180,E1 -1527.258,E2 -1527.258} C_VEL
LIN {X 0,Y 587.141,Z 557.205,A -85,B 0,C 180,E1 -1527.945,E2 -1527.945} C_VEL
LIN {X 0,Y 587.14,Z 558.786,A -85,B 0,C 180,E1 -1529.317,E2 -1529.317} C_VEL
LIN {X 0,Y 587.137,Z 559,A -85,B 0,C 180,E1 -1530.003,E2 -1530.003} C_VEL
LIN {X 0,Y 587.147,Z 558.182,A -85,B 0,C 180,E1 -1531.374,E2 -1531.374} C_VEL
LIN {X 0,Y 587.141,Z 557.197,A -85,B 0,C 180,E1 -1532.06,E2 -1532.06} C_VEL
LIN {X 0,Y 587.132,Z 555.804,A -85,B 0,C 180,E1 -1532.747,E2 -1532.747} C_VEL
LIN {X 0,Y 587.213,Z 552.888,A -85,B 0,C 180,E1 -1533.777,E2 -1533.777} C_VEL
LIN {X 0,Y 587.147,Z 548.94,A -85,B 0,C 180,E1 -1534.809,E2 -1534.809} C_VEL
LIN {X 0,Y 587.218,Z 542.864,A -85,B 0,C 180,E1 -1536.014,E2 -1536.014} C_VEL
LIN {X 0,Y 587.247,Z 536.22,A -85,B 0,C 180,E1 -1537.048,E2 -1537.048} C_VEL
LIN {X 0,Y 587.299,Z 527.97,A -85,B 0,C 180,E1 -1538.085,E2 -1538.085} C_VEL
LIN {X 0,Y 587.344,Z 519.513,A -85,B 0,C 180,E1 -1538.951,E2 -1538.951} C_VEL
LIN {X 0,Y 587.422,Z 509.065,A -85,B 0,C 180,E1 -1539.818,E2 -1539.818} C_VEL
LIN {X 0,Y 587.48,Z 498.722,A -85,B 0,C 180,E1 -1540.514,E2 -1540.514} C_VEL
LIN {X 0,Y 587.535,Z 487.115,A -85,B 0,C 180,E1 -1541.135,E2 -1541.135} C_VEL
LIN {X 0,Y 587.628,Z 474.628,A -85,B 0,C 180,E1 -1541.638,E2 -1541.638} C_VEL
LIN {X 0,Y 587.72,Z 461.345,A -85,B 0,C 180,E1 -1542.016,E2 -1542.016} C_VEL
LIN {X 0,Y 587.5,Z 453.463,A -85,B 0,C 180,E1 -1542.174,E2 -1542.174} C_VEL
LIN {X 0,Y 587.207,Z 451.522,A -85,B 0,C 180,E1 -1542.224,E2 -1542.224} C_VEL
LIN {X 0,Y 587.261,Z 441.428,A -85,B 0,C 180,E1 -1544.912,E2 -1544.912} C_VEL
LIN {X 0,Y 587.304,Z 430.837,A -85,B 0,C 180,E1 -1547.769,E2 -1547.769} C_VEL
LIN {X 0,Y 587.379,Z 420.246,A -85,B 0,C 180,E1 -1550.671,E2 -1550.671} C_VEL
LIN {X 0,Y 587.39,Z 410.979,A -85,B 0,C 180,E1 -1553.258,E2 -1553.258} C_VEL
LIN {X 0,Y 587.47,Z 401.847,A -85,B 0,C 180,E1 -1555.854,E2 -1555.854} C_VEL
LIN {X 0,Y 587.466,Z 392.385,A -85,B 0,C 180,E1 -1558.591,E2 -1558.591} C_VEL
LIN {X 0,Y 587.534,Z 384.312,A -85,B 0,C 180,E1 -1560.956,E2 -1560.956} C_VEL
LIN {X 0,Y 587.671,Z 375.165,A -85,B 0,C 180,E1 -1563.788,E2 -1563.788} C_VEL
LIN {X 0,Y 587.583,Z 368.66,A -85,B 0,C 180,E1 -1565.881,E2 -1565.881} C_VEL
LIN {X 0,Y 587.338,Z 367.327,A -85,B 0,C 180,E1 -1566.37,E2 -1566.37} C_VEL
LIN {X 0,Y 587.323,Z 367.328,A -85,B 0,C 180,E1 -1568.94,E2 -1568.94} C_VEL
LIN {X 0,Y 587.342,Z 367.323,A -85,B 0,C 180,E1 -1571.158,E2 -1571.158} C_VEL
LIN {X 0,Y 587.323,Z 367.326,A -85,B 0,C 180,E1 -1574.112,E2 -1574.112} C_VEL
LIN {X 0,Y 587.301,Z 367.33,A -85,B 0,C 180,E1 -1576.992,E2 -1576.992} C_VEL
LIN {X 0,Y 587.32,Z 367.329,A -85,B 0,C 180,E1 -1579.746,E2 -1579.746} C_VEL
LIN {X 0,Y 587.349,Z 367.324,A -85,B 0,C 180,E1 -1582.392,E2 -1582.392} C_VEL
LIN {X 0,Y 587.348,Z 367.323,A -85,B 0,C 180,E1 -1585.654,E2 -1585.654} C_VEL
LIN {X 0,Y 587.342,Z 367.325,A -85,B 0,C 180,E1 -1588.231,E2 -1588.231} C_VEL
LIN {X 0,Y 587.357,Z 367.324,A -85,B 0,C 180,E1 -1590.867,E2 -1590.867} C_VEL
LIN {X 0,Y 587.312,Z 367.327,A -85,B 0,C 180,E1 -1593.83,E2 -1593.83} C_VEL
LIN {X 0,Y 587.337,Z 367.328,A -85,B 0,C 180,E1 -1595.993,E2 -1595.993} C_VEL
LIN {X 0,Y 587.341,Z 367.325,A -85,B 0,C 180,E1 -1598.962,E2 -1598.962} C_VEL
LIN {X 0,Y 587.353,Z 367.324,A -85,B 0,C 180,E1 -1601.151,E2 -1601.151} C_VEL
LIN {X 0,Y 587.324,Z 367.33,A -85,B 0,C 180,E1 -1604.024,E2 -1604.024} C_VEL
LIN {X 0,Y 587.346,Z 367.322,A -85,B 0,C 180,E1 -1606.153,E2 -1606.153} C_VEL
LIN {X 0,Y 587.349,Z 367.323,A -85,B 0,C 180,E1 -1608.962,E2 -1608.962} C_VEL
LIN {X 0,Y 587.348,Z 367.323,A -85,B 0,C 180,E1 -1611.744,E2 -1611.744} C_VEL
LIN {X 0,Y 587.356,Z 367.323,A -85,B 0,C 180,E1 -1614.506,E2 -1614.506} C_VEL
LIN {X 0,Y 587.383,Z 367.32,A -85,B 0,C 180,E1 -1617.256,E2 -1617.256} C_VEL
LIN {X 0,Y 587.385,Z 367.32,A -85,B 0,C 180,E1 -1619.999,E2 -1619.999} C_VEL
LIN {X 0,Y 587.368,Z 367.323,A -85,B 0,C 180,E1 -1622.743,E2 -1622.743} C_VEL
LIN {X 0,Y 587.356,Z 367.326,A -85,B 0,C 180,E1 -1625.492,E2 -1625.492} C_VEL
LIN {X 0,Y 587.333,Z 367.329,A -85,B 0,C 180,E1 -1628.255,E2 -1628.255} C_VEL
LIN {X 0,Y 587.356,Z 367.323,A -85,B 0,C 180,E1 -1631.133,E2 -1631.133} C_VEL
LIN {X 0,Y 587.35,Z 367.324,A -85,B 0,C 180,E1 -1633.845,E2 -1633.845} C_VEL
LIN {X 0,Y 587.366,Z 367.32,A -85,B 0,C 180,E1 -1636.817,E2 -1636.817} C_VEL
LIN {X 0,Y 587.303,Z 367.328,A -85,B 0,C 180,E1 -1638.293,E2 -1638.293} C_VEL
LIN {X 0,Y 586.664,Z 367.411,A -85,B 0,C 180,E1 -1638.865,E2 -1638.865} C_VEL
LIN {X 0,Y 583.848,Z 367.764,A -85,B 0,C 180,E1 -1639.794,E2 -1639.794} C_VEL
LIN {X 0,Y 581.44,Z 368.064,A -85,B 0,C 180,E1 -1640.541,E2 -1640.541} C_VEL
LIN {X 0,Y 580.385,Z 368.193,A -85,B 0,C 180,E1 -1641.117,E2 -1641.117} C_VEL
LIN {X 0,Y 580.289,Z 368.203,A -85,B 0,C 180,E1 -1641.313,E2 -1641.313} C_VEL
LIN {X 0,Y 580.27,Z 368.204,A -85,B 0,C 180,E1 -1643.558,E2 -1643.558} C_VEL
LIN {X 0,Y 580.288,Z 368.204,A -85,B 0,C 180,E1 -1645.848,E2 -1645.848} C_VEL
LIN {X 0,Y 580.297,Z 368.201,A -85,B 0,C 180,E1 -1648.975,E2 -1648.975} C_VEL
LIN {X 0,Y 580.306,Z 368.201,A -85,B 0,C 180,E1 -1652.029,E2 -1652.029} C_VEL
LIN {X 0,Y 580.294,Z 368.202,A -85,B 0,C 180,E1 -1654.695,E2 -1654.695} C_VEL
LIN {X 0,Y 580.292,Z 368.202,A -85,B 0,C 180,E1 -1657.268,E2 -1657.268} C_VEL
LIN {X 0,Y 580.289,Z 368.205,A -85,B 0,C 180,E1 -1660.268,E2 -1660.268} C_VEL
LIN {X 0,Y 580.277,Z 368.204,A -85,B 0,C 180,E1 -1662.705,E2 -1662.705} C_VEL
LIN {X 0,Y 580.258,Z 368.209,A -85,B 0,C 180,E1 -1665.609,E2 -1665.609} C_VEL
LIN {X 0,Y 580.272,Z 368.206,A -85,B 0,C 180,E1 -1668.229,E2 -1668.229} C_VEL
LIN {X 0,Y 580.286,Z 368.205,A -85,B 0,C 180,E1 -1670.964,E2 -1670.964} C_VEL
LIN {X 0,Y 580.258,Z 368.208,A -85,B 0,C 180,E1 -1673.594,E2 -1673.594} C_VEL
LIN {X 0,Y 580.309,Z 368.2,A -85,B 0,C 180,E1 -1676.143,E2 -1676.143} C_VEL
LIN {X 0,Y 580.286,Z 368.202,A -85,B 0,C 180,E1 -1678.613,E2 -1678.613} C_VEL
LIN {X 0,Y 580.288,Z 368.202,A -85,B 0,C 180,E1 -1681.022,E2 -1681.022} C_VEL
LIN {X 0,Y 580.293,Z 368.201,A -85,B 0,C 180,E1 -1683.664,E2 -1683.664} C_VEL
LIN {X 0,Y 580.302,Z 368.202,A -85,B 0,C 180,E1 -1685.682,E2 -1685.682} C_VEL
LIN {X 0,Y 580.271,Z 368.204,A -85,B 0,C 180,E1 -1687.945,E2 -1687.945} C_VEL
LIN {X 0,Y 580.297,Z 368.202,A -85,B 0,C 180,E1 -1690.911,E2 -1690.911} C_VEL
LIN {X 0,Y 580.266,Z 368.208,A -85,B 0,C 180,E1 -1693.823,E2 -1693.823} C_VEL
LIN {X 0,Y 580.324,Z 368.197,A -85,B 0,C 180,E1 -1695.981,E2 -1695.981} C_VEL
LIN {X 0,Y 580.301,Z 368.201,A -85,B 0,C 180,E1 -1698.825,E2 -1698.825} C_VEL
LIN {X 0,Y 580.321,Z 368.199,A -85,B 0,C 180,E1 -1701.642,E2 -1701.642} C_VEL
LIN {X 0,Y 580.331,Z 368.199,A -85,B 0,C 180,E1 -1704.438,E2 -1704.438} C_VEL
LIN {X 0,Y 580.343,Z 368.195,A -85,B 0,C 180,E1 -1707.915,E2 -1707.915} C_VEL
LIN {X 0,Y 580.345,Z 368.195,A -85,B 0,C 180,E1 -1710.691,E2 -1710.691} C_VEL
LIN {X 0,Y 580.336,Z 368.199,A -85,B 0,C 180,E1 -1712.774,E2 -1712.774} C_VEL
LIN {X 0,Y 580.33,Z 368.199,A -85,B 0,C 180,E1 -1715.557,E2 -1715.557} C_VEL
LIN {X 0,Y 580.318,Z 368.199,A -85,B 0,C 180,E1 -1718.353,E2 -1718.353} C_VEL
LIN {X 0,Y 580.321,Z 368.198,A -85,B 0,C 180,E1 -1721.206,E2 -1721.206} C_VEL
LIN {X 0,Y 580.302,Z 368.201,A -85,B 0,C 180,E1 -1724.337,E2 -1724.337} C_VEL
LIN {X 0,Y 580.296,Z 368.201,A -85,B 0,C 180,E1 -1726.911,E2 -1726.911} C_VEL
LIN {X 0,Y 580.292,Z 368.203,A -85,B 0,C 180,E1 -1729.819,E2 -1729.819} C_VEL
LIN {X 0,Y 580.296,Z 368.205,A -85,B 0,C 180,E1 -1732.799,E2 -1732.799} C_VEL
LIN {X 0,Y 580.294,Z 368.201,A -85,B 0,C 180,E1 -1735.077,E2 -1735.077} C_VEL
LIN {X 0,Y 580.196,Z 368.218,A -85,B 0,C 180,E1 -1737.403,E2 -1737.403} C_VEL
LIN {X 0,Y 580.154,Z 368.732,A -85,B 0,C 180,E1 -1738.189,E2 -1738.189} C_VEL
LIN {X 0,Y 580.145,Z 371.628,A -85,B 0,C 180,E1 -1740.673,E2 -1740.673} C_VEL
LIN {X 0,Y 580.099,Z 374.676,A -85,B 0,C 180,E1 -1743.287,E2 -1743.287} C_VEL
LIN {X 0,Y 580.083,Z 378.333,A -85,B 0,C 180,E1 -1746.413,E2 -1746.413} C_VEL
LIN {X 0,Y 580.052,Z 381.728,A -85,B 0,C 180,E1 -1749.157,E2 -1749.157} C_VEL
LIN {X 0,Y 580.067,Z 385.108,A -85,B 0,C 180,E1 -1751.783,E2 -1751.783} C_VEL
LIN {X 0,Y 580.068,Z 388.851,A -85,B 0,C 180,E1 -1754.64,E2 -1754.64} C_VEL
LIN {X 0,Y 580.056,Z 392.856,A -85,B 0,C 180,E1 -1757.647,E2 -1757.647} C_VEL
LIN {X 0,Y 580.045,Z 395.739,A -85,B 0,C 180,E1 -1759.752,E2 -1759.752} C_VEL
LIN {X 0,Y 580.778,Z 401.671,A -85,B 0,C 180,E1 -1759.891,E2 -1759.891} C_VEL
LIN {X 0,Y 580.668,Z 415.286,A -85,B 0,C 180,E1 -1760.288,E2 -1760.288} C_VEL
LIN {X 0,Y 580.585,Z 427.094,A -85,B 0,C 180,E1 -1760.774,E2 -1760.774} C_VEL
LIN {X 0,Y 580.473,Z 439.108,A -85,B 0,C 180,E1 -1761.427,E2 -1761.427} C_VEL
LIN {X 0,Y 580.398,Z 450.338,A -85,B 0,C 180,E1 -1762.203,E2 -1762.203} C_VEL
LIN {X 0,Y 580.308,Z 460.278,A -85,B 0,C 180,E1 -1763.058,E2 -1763.058} C_VEL
LIN {X 0,Y 580.231,Z 468.7,A -85,B 0,C 180,E1 -1763.946,E2 -1763.946} C_VEL
LIN {X 0,Y 580.164,Z 475.958,A -85,B 0,C 180,E1 -1764.873,E2 -1764.873} C_VEL
LIN {X 0,Y 580.125,Z 481.913,A -85,B 0,C 180,E1 -1765.793,E2 -1765.793} C_VEL
LIN {X 0,Y 580.095,Z 487.976,A -85,B 0,C 180,E1 -1766.964,E2 -1766.964} C_VEL
LIN {X 0,Y 580.064,Z 492.114,A -85,B 0,C 180,E1 -1767.999,E2 -1767.999} C_VEL
LIN {X 0,Y 580.068,Z 495.958,A -85,B 0,C 180,E1 -1769.334,E2 -1769.334} C_VEL
LIN {X 0,Y 580.049,Z 498.264,A -85,B 0,C 180,E1 -1770.726,E2 -1770.726} C_VEL
LIN {X 0,Y 580.026,Z 498.975,A -85,B 0,C 180,E1 -1772.183,E2 -1772.183} C_VEL
LIN {X 0,Y 580.037,Z 498.261,A -85,B 0,C 180,E1 -1773.366,E2 -1773.366} C_VEL
LIN {X 0,Y 580.029,Z 497.181,A -85,B 0,C 180,E1 -1774.139,E2 -1774.139} C_VEL
LIN {X 0,Y 580.065,Z 494.555,A -85,B 0,C 180,E1 -1775.315,E2 -1775.315} C_VEL
LIN {X 0,Y 580.09,Z 490.883,A -85,B 0,C 180,E1 -1776.435,E2 -1776.435} C_VEL
LIN {X 0,Y 580.122,Z 485.885,A -85,B 0,C 180,E1 -1777.567,E2 -1777.567} C_VEL
LIN {X 0,Y 580.165,Z 479.499,A -85,B 0,C 180,E1 -1778.691,E2 -1778.691} C_VEL
LIN {X 0,Y 580.215,Z 471.525,A -85,B 0,C 180,E1 -1779.806,E2 -1779.806} C_VEL
LIN {X 0,Y 580.28,Z 462.216,A -85,B 0,C 180,E1 -1780.841,E2 -1780.841} C_VEL
LIN {X 0,Y 580.403,Z 452.176,A -85,B 0,C 180,E1 -1781.742,E2 -1781.742} C_VEL
LIN {X 0,Y 580.417,Z 442.181,A -85,B 0,C 180,E1 -1782.471,E2 -1782.471} C_VEL
LIN {X 0,Y 580.516,Z 431.247,A -85,B 0,C 180,E1 -1783.11,E2 -1783.11} C_VEL
LIN {X 0,Y 580.63,Z 419.196,A -85,B 0,C 180,E1 -1783.656,E2 -1783.656} C_VEL
LIN {X 0,Y 580.749,Z 406.158,A -85,B 0,C 180,E1 -1784.088,E2 -1784.088} C_VEL
LIN {X 0,Y 580.557,Z 399.042,A -85,B 0,C 180,E1 -1784.263,E2 -1784.263} C_VEL
LIN {X 0,Y 580.038,Z 395.724,A -85,B 0,C 180,E1 -1784.338,E2 -1784.338} C_VEL
LIN {X 0,Y 580.038,Z 391.571,A -85,B 0,C 180,E1 -1787.403,E2 -1787.403} C_VEL
LIN {X 0,Y 580.022,Z 388.749,A -85,B 0,C 180,E1 -1789.529,E2 -1789.529} C_VEL
LIN {X 0,Y 580.048,Z 385.064,A -85,B 0,C 180,E1 -1792.342,E2 -1792.342} C_VEL
LIN {X 0,Y 580.066,Z 381.47,A -85,B 0,C 180,E1 -1795.135,E2 -1795.135} C_VEL
LIN {X 0,Y 580.042,Z 378.873,A -85,B 0,C 180,E1 -1797.223,E2 -1797.223} C_VEL
LIN {X 0,Y 580.157,Z 376.7,A -85,B 0,C 180,E1 -1799.307,E2 -1799.307} C_VEL
LIN {X 0,Y 580.175,Z 374.367,A -85,B 0,C 180,E1 -1801.389,E2 -1801.389} C_VEL
LIN {X 0,Y 580.206,Z 371.112,A -85,B 0,C 180,E1 -1804.168,E2 -1804.168} C_VEL
LIN {X 0,Y 580.225,Z 368.215,A -85,B 0,C 180,E1 -1806.71,E2 -1806.71} C_VEL
LIN {X 0,Y 580.267,Z 368.206,A -85,B 0,C 180,E1 -1809.06,E2 -1809.06} C_VEL
LIN {X 0,Y 580.344,Z 368.194,A -85,B 0,C 180,E1 -1811.234,E2 -1811.234} C_VEL
LIN {X 0,Y 580.278,Z 368.203,A -85,B 0,C 180,E1 -1814.341,E2 -1814.341} C_VEL
LIN {X 0,Y 580.307,Z 368.198,A -85,B 0,C 180,E1 -1816.926,E2 -1816.926} C_VEL
LIN {X 0,Y 580.282,Z 368.202,A -85,B 0,C 180,E1 -1819.824,E2 -1819.824} C_VEL
LIN {X 0,Y 580.322,Z 368.196,A -85,B 0,C 180,E1 -1822.802,E2 -1822.802} C_VEL
LIN {X 0,Y 580.265,Z 368.204,A -85,B 0,C 180,E1 -1825.851,E2 -1825.851} C_VEL
LIN {X 0,Y 580.284,Z 368.206,A -85,B 0,C 180,E1 -1828.187,E2 -1828.187} C_VEL
LIN {X 0,Y 580.273,Z 368.204,A -85,B 0,C 180,E1 -1830.701,E2 -1830.701} C_VEL
LIN {X 0,Y 580.279,Z 368.202,A -85,B 0,C 180,E1 -1833.32,E2 -1833.32} C_VEL
LIN {X 0,Y 580.305,Z 368.201,A -85,B 0,C 180,E1 -1835.771,E2 -1835.771} C_VEL
LIN {X 0,Y 580.262,Z 368.206,A -85,B 0,C 180,E1 -1838.149,E2 -1838.149} C_VEL
LIN {X 0,Y 580.3,Z 368.2,A -85,B 0,C 180,E1 -1840.844,E2 -1840.844} C_VEL
LIN {X 0,Y 580.267,Z 368.204,A -85,B 0,C 180,E1 -1843.659,E2 -1843.659} C_VEL
LIN {X 0,Y 580.272,Z 368.203,A -85,B 0,C 180,E1 -1846.61,E2 -1846.61} C_VEL
LIN {X 0,Y 580.296,Z 368.203,A -85,B 0,C 180,E1 -1849.161,E2 -1849.161} C_VEL
LIN {X 0,Y 580.276,Z 368.209,A -85,B 0,C 180,E1 -1851.929,E2 -1851.929} C_VEL
LIN {X 0,Y 580.318,Z 368.286,A -85,B 0,C 180,E1 -1853.413,E2 -1853.413} C_VEL
LIN {X 0,Y 580.737,Z 372.539,A -85,B 0,C 180,E1 -1854.916,E2 -1854.916} C_VEL
LIN {X 0,Y 580.63,Z 380.225,A -85,B 0,C 180,E1 -1857.414,E2 -1857.414} C_VEL
LIN {X 0,Y 580.529,Z 389.567,A -85,B 0,C 180,E1 -1860.245,E2 -1860.245} C_VEL
LIN {X 0,Y 580.42,Z 399.031,A -85,B 0,C 180,E1 -1862.999,E2 -1862.999} C_VEL
LIN {X 0,Y 580.415,Z 406.816,A -85,B 0,C 180,E1 -1865.251,E2 -1865.251} C_VEL
LIN {X 0,Y 580.365,Z 416.294,A -85,B 0,C 180,E1 -1867.955,E2 -1867.955} C_VEL
LIN {X 0,Y 580.258,Z 426.69,A -85,B 0,C 180,E1 -1870.861,E2 -1870.861} C_VEL
LIN {X 0,Y 580.22,Z 437.475,A -85,B 0,C 180,E1 -1873.827,E2 -1873.827} C_VEL
LIN {X 0,Y 580.183,Z 448.066,A -85,B 0,C 180,E1 -1876.697,E2 -1876.697} C_VEL
LIN {X 0,Y 580.141,Z 451.583,A -85,B 0,C 180,E1 -1877.641,E2 -1877.641} C_VEL
LIN {X 0,Y 580.804,Z 457.384,A -85,B 0,C 180,E1 -1877.755,E2 -1877.755} C_VEL
LIN {X 0,Y 580.732,Z 470.6,A -85,B 0,C 180,E1 -1878.086,E2 -1878.086} C_VEL
LIN {X 0,Y 580.614,Z 482.385,A -85,B 0,C 180,E1 -1878.518,E2 -1878.518} C_VEL
LIN {X 0,Y 580.5,Z 494.264,A -85,B 0,C 180,E1 -1879.099,E2 -1879.099} C_VEL
LIN {X 0,Y 580.457,Z 505.522,A -85,B 0,C 180,E1 -1879.803,E2 -1879.803} C_VEL
LIN {X 0,Y 580.351,Z 515.68,A -85,B 0,C 180,E1 -1880.594,E2 -1880.594} C_VEL
LIN {X 0,Y 580.278,Z 524.813,A -85,B 0,C 180,E1 -1881.471,E2 -1881.471} C_VEL
LIN {X 0,Y 580.197,Z 533.712,A -85,B 0,C 180,E1 -1882.521,E2 -1882.521} C_VEL
LIN {X 0,Y 580.119,Z 540.474,A -85,B 0,C 180,E1 -1883.506,E2 -1883.506} C_VEL
LIN {X 0,Y 580.139,Z 545.694,A -85,B 0,C 180,E1 -1884.441,E2 -1884.441} C_VEL
LIN {X 0,Y 580.108,Z 550.383,A -85,B 0,C 180,E1 -1885.486,E2 -1885.486} C_VEL
LIN {X 0,Y 580.122,Z 553.965,A -85,B 0,C 180,E1 -1886.53,E2 -1886.53} C_VEL
LIN {X 0,Y 580.043,Z 555.815,A -85,B 0,C 180,E1 -1887.225,E2 -1887.225} C_VEL
LIN {X 0,Y 580.04,Z 557.204,A -85,B 0,C 180,E1 -1887.919,E2 -1887.919} C_VEL
LIN {X 0,Y 580.04,Z 558.786,A -85,B 0,C 180,E1 -1889.308,E2 -1889.308} C_VEL
LIN {X 0,Y 580.037,Z 559,A -85,B 0,C 180,E1 -1890.003,E2 -1890.003} C_VEL
LIN {X 0,Y 580.047,Z 558.183,A -85,B 0,C 180,E1 -1891.391,E2 -1891.391} C_VEL
LIN {X 0,Y 580.04,Z 557.197,A -85,B 0,C 180,E1 -1892.086,E2 -1892.086} C_VEL
LIN {X 0,Y 580.043,Z 555.804,A -85,B 0,C 180,E1 -1892.78,E2 -1892.78} C_VEL
LIN {X 0,Y 580.11,Z 552.888,A -85,B 0,C 180,E1 -1893.823,E2 -1893.823} C_VEL
LIN {X 0,Y 580.053,Z 548.939,A -85,B 0,C 180,E1 -1894.868,E2 -1894.868} C_VEL
LIN {X 0,Y 580.141,Z 542.864,A -85,B 0,C 180,E1 -1896.087,E2 -1896.087} C_VEL
LIN {X 0,Y 580.187,Z 536.22,A -85,B 0,C 180,E1 -1897.135,E2 -1897.135} C_VEL
LIN {X 0,Y 580.247,Z 527.971,A -85,B 0,C 180,E1 -1898.184,E2 -1898.184} C_VEL
LIN {X 0,Y 580.309,Z 519.513,A -85,B 0,C 180,E1 -1899.061,E2 -1899.061} C_VEL
LIN {X 0,Y 580.424,Z 509.066,A -85,B 0,C 180,E1 -1899.938,E2 -1899.938} C_VEL
LIN {X 0,Y 580.5,Z 498.721,A -85,B 0,C 180,E1 -1900.642,E2 -1900.642} C_VEL
LIN {X 0,Y 580.568,Z 487.546,A -85,B 0,C 180,E1 -1901.25,E2 -1901.25} C_VEL
LIN {X 0,Y 580.669,Z 475.702,A -85,B 0,C 180,E1 -1901.743,E2 -1901.743} C_VEL
LIN {X 0,Y 580.778,Z 462.259,A -85,B 0,C 180,E1 -1902.139,E2 -1902.139} C_VEL
LIN {X 0,Y 580.6,Z 454.365,A -85,B 0,C 180,E1 -1902.307,E2 -1902.307} C_VEL
LIN {X 0,Y 580.131,Z 451.522,A -85,B 0,C 180,E1 -1902.375,E2 -1902.375} C_VEL
LIN {X 0,Y 580.221,Z 441.428,A -85,B 0,C 180,E1 -1905.097,E2 -1905.097} C_VEL
LIN {X 0,Y 580.257,Z 430.837,A -85,B 0,C 180,E1 -1907.992,E2 -1907.992} C_VEL
LIN {X 0,Y 580.329,Z 420.492,A -85,B 0,C 180,E1 -1910.865,E2 -1910.865} C_VEL
LIN {X 0,Y 580.385,Z 410.979,A -85,B 0,C 180,E1 -1913.555,E2 -1913.555} C_VEL
LIN {X 0,Y 580.454,Z 401.237,A -85,B 0,C 180,E1 -1916.366,E2 -1916.366} C_VEL
LIN {X 0,Y 580.472,Z 392.287,A -85,B 0,C 180,E1 -1918.968,E2 -1918.968} C_VEL
LIN {X 0,Y 580.587,Z 384.293,A -85,B 0,C 180,E1 -1921.369,E2 -1921.369} C_VEL
LIN {X 0,Y 580.724,Z 376.436,A -85,B 0,C 180,E1 -1923.83,E2 -1923.83} C_VEL
LIN {X 0,Y 580.667,Z 370.374,A -85,B 0,C 180,E1 -1925.813,E2 -1925.813} C_VEL
LIN {X 0,Y 580.302,Z 368.205,A -85,B 0,C 180,E1 -1926.593,E2 -1926.593} C_VEL
LIN {X 0,Y 580.299,Z 368.205,A -85,B 0,C 180,E1 -1929.185,E2 -1929.185} C_VEL
LIN {X 0,Y 580.264,Z 368.209,A -85,B 0,C 180,E1 -1931.772,E2 -1931.772} C_VEL
LIN {X 0,Y 580.259,Z 368.209,A -85,B 0,C 180,E1 -1934.629,E2 -1934.629} C_VEL
LIN {X 0,Y 580.275,Z 368.204,A -85,B 0,C 180,E1 -1937.631,E2 -1937.631} C_VEL
LIN {X 0,Y 580.289,Z 368.205,A -85,B 0,C 180,E1 -1940.066,E2 -1940.066} C_VEL
LIN {X 0,Y 580.288,Z 368.202,A -85,B 0,C 180,E1 -1943.069,E2 -1943.069} C_VEL
LIN {X 0,Y 580.29,Z 368.202,A -85,B 0,C 180,E1 -1946.143,E2 -1946.143} C_VEL
LIN {X 0,Y 580.275,Z 368.203,A -85,B 0,C 180,E1 -1948.614,E2 -1948.614} C_VEL
LIN {X 0,Y 580.3,Z 368.201,A -85,B 0,C 180,E1 -1951.024,E2 -1951.024} C_VEL
LIN {X 0,Y 580.266,Z 368.204,A -85,B 0,C 180,E1 -1954.149,E2 -1954.149} C_VEL
LIN {X 0,Y 580.28,Z 368.203,A -85,B 0,C 180,E1 -1956.442,E2 -1956.442} C_VEL
LIN {X 0,Y 580.279,Z 368.203,A -85,B 0,C 180,E1 -1959.437,E2 -1959.437} C_VEL
LIN {X 0,Y 580.263,Z 368.206,A -85,B 0,C 180,E1 -1961.644,E2 -1961.644} C_VEL
LIN {X 0,Y 580.279,Z 368.205,A -85,B 0,C 180,E1 -1963.825,E2 -1963.825} C_VEL
LIN {X 0,Y 580.27,Z 368.208,A -85,B 0,C 180,E1 -1966.695,E2 -1966.695} C_VEL
LIN {X 0,Y 580.315,Z 368.199,A -85,B 0,C 180,E1 -1968.827,E2 -1968.827} C_VEL
LIN {X 0,Y 580.317,Z 368.199,A -85,B 0,C 180,E1 -1971.643,E2 -1971.643} C_VEL
LIN {X 0,Y 580.274,Z 368.205,A -85,B 0,C 180,E1 -1973.742,E2 -1973.742} C_VEL
LIN {X 0,Y 580.268,Z 368.206,A -85,B 0,C 180,E1 -1975.832,E2 -1975.832} C_VEL
LIN {X 0,Y 580.326,Z 368.197,A -85,B 0,C 180,E1 -1977.917,E2 -1977.917} C_VEL
LIN {X 0,Y 580.365,Z 368.193,A -85,B 0,C 180,E1 -1980.693,E2 -1980.693} C_VEL
LIN {X 0,Y 580.276,Z 368.203,A -85,B 0,C 180,E1 -1983.471,E2 -1983.471} C_VEL
LIN {X 0,Y 580.32,Z 368.202,A -85,B 0,C 180,E1 -1985.559,E2 -1985.559} C_VEL
LIN {X 0,Y 580.306,Z 368.203,A -85,B 0,C 180,E1 -1988.356,E2 -1988.356} C_VEL
LIN {X 0,Y 580.308,Z 368.201,A -85,B 0,C 180,E1 -1991.19,E2 -1991.19} C_VEL
LIN {X 0,Y 580.31,Z 368.2,A -85,B 0,C 180,E1 -1994.017,E2 -1994.017} C_VEL
LIN {X 0,Y 580.319,Z 368.198,A -85,B 0,C 180,E1 -1996.913,E2 -1996.913} C_VEL
LIN {X 0,Y 580.289,Z 368.202,A -85,B 0,C 180,E1 -1999.822,E2 -1999.822} C_VEL
LIN {X 0,Y 580.289,Z 368.203,A -85,B 0,C 180,E1 -2001.313,E2 -2001.313} C_VEL
LIN {X 0,Y 579.586,Z 368.291,A -85,B 0,C 180,E1 -2001.892,E2 -2001.892} C_VEL
LIN {X 0,Y 576.705,Z 368.651,A -85,B 0,C 180,E1 -2002.832,E2 -2002.832} C_VEL
LIN {X 0,Y 574.31,Z 368.947,A -85,B 0,C 180,E1 -2003.588,E2 -2003.588} C_VEL
LIN {X 0,Y 573.314,Z 369.073,A -85,B 0,C 180,E1 -2004.172,E2 -2004.172} C_VEL
LIN {X 0,Y 573.249,Z 369.078,A -85,B 0,C 180,E1 -2004.369,E2 -2004.369} C_VEL
LIN {X 0,Y 573.214,Z 369.087,A -85,B 0,C 180,E1 -2006.977,E2 -2006.977} C_VEL
LIN {X 0,Y 573.247,Z 369.082,A -85,B 0,C 180,E1 -2009.486,E2 -2009.486} C_VEL
LIN {X 0,Y 573.258,Z 369.079,A -85,B 0,C 180,E1 -2012.644,E2 -2012.644} C_VEL
LIN {X 0,Y 573.21,Z 369.086,A -85,B 0,C 180,E1 -2015.187,E2 -2015.187} C_VEL
LIN {X 0,Y 573.236,Z 369.084,A -85,B 0,C 180,E1 -2017.806,E2 -2017.806} C_VEL
LIN {X 0,Y 573.248,Z 369.082,A -85,B 0,C 180,E1 -2020.524,E2 -2020.524} C_VEL
LIN {X 0,Y 573.213,Z 369.084,A -85,B 0,C 180,E1 -2023.36,E2 -2023.36} C_VEL
LIN {X 0,Y 573.239,Z 369.08,A -85,B 0,C 180,E1 -2026.33,E2 -2026.33} C_VEL
LIN {X 0,Y 573.247,Z 369.08,A -85,B 0,C 180,E1 -2029.473,E2 -2029.473} C_VEL
LIN {X 0,Y 573.23,Z 369.083,A -85,B 0,C 180,E1 -2032.19,E2 -2032.19} C_VEL
LIN {X 0,Y 573.252,Z 369.082,A -85,B 0,C 180,E1 -2035.225,E2 -2035.225} C_VEL
LIN {X 0,Y 573.255,Z 369.081,A -85,B 0,C 180,E1 -2037.77,E2 -2037.77} C_VEL
LIN {X 0,Y 573.256,Z 369.081,A -85,B 0,C 180,E1 -2040.632,E2 -2040.632} C_VEL
LIN {X 0,Y 573.252,Z 369.081,A -85,B 0,C 180,E1 -2043.022,E2 -2043.022} C_VEL
LIN {X 0,Y 573.276,Z 369.075,A -85,B 0,C 180,E1 -2045.364,E2 -2045.364} C_VEL
LIN {X 0,Y 573.228,Z 369.084,A -85,B 0,C 180,E1 -2048.417,E2 -2048.417} C_VEL
LIN {X 0,Y 573.268,Z 369.077,A -85,B 0,C 180,E1 -2050.729,E2 -2050.729} C_VEL
LIN {X 0,Y 573.24,Z 369.081,A -85,B 0,C 180,E1 -2053.619,E2 -2053.619} C_VEL
LIN {X 0,Y 573.271,Z 369.076,A -85,B 0,C 180,E1 -2055.805,E2 -2055.805} C_VEL
LIN {X 0,Y 573.26,Z 369.078,A -85,B 0,C 180,E1 -2058.743,E2 -2058.743} C_VEL
LIN {X 0,Y 573.278,Z 369.075,A -85,B 0,C 180,E1 -2061.538,E2 -2061.538} C_VEL
LIN {X 0,Y 573.298,Z 369.074,A -85,B 0,C 180,E1 -2064.369,E2 -2064.369} C_VEL
LIN {X 0,Y 573.313,Z 369.071,A -85,B 0,C 180,E1 -2067.89,E2 -2067.89} C_VEL
LIN {X 0,Y 573.317,Z 369.07,A -85,B 0,C 180,E1 -2070.7,E2 -2070.7} C_VEL
LIN {X 0,Y 573.301,Z 369.075,A -85,B 0,C 180,E1 -2072.808,E2 -2072.808} C_VEL
LIN {X 0,Y 573.297,Z 369.075,A -85,B 0,C 180,E1 -2075.625,E2 -2075.625} C_VEL
LIN {X 0,Y 573.274,Z 369.076,A -85,B 0,C 180,E1 -2078.457,E2 -2078.457} C_VEL
LIN {X 0,Y 573.287,Z 369.074,A -85,B 0,C 180,E1 -2081.309,E2 -2081.309} C_VEL
LIN {X 0,Y 573.268,Z 369.078,A -85,B 0,C 180,E1 -2084.422,E2 -2084.422} C_VEL
LIN {X 0,Y 573.244,Z 369.08,A -85,B 0,C 180,E1 -2087.109,E2 -2087.109} C_VEL
LIN {X 0,Y 573.238,Z 369.084,A -85,B 0,C 180,E1 -2090.074,E2 -2090.074} C_VEL
LIN {X 0,Y 573.253,Z 369.079,A -85,B 0,C 180,E1 -2093.151,E2 -2093.151} C_VEL
LIN {X 0,Y 573.242,Z 369.083,A -85,B 0,C 180,E1 -2095.407,E2 -2095.407} C_VEL
LIN {X 0,Y 573.1,Z 369.145,A -85,B 0,C 180,E1 -2098.002,E2 -2098.002} C_VEL
LIN {X 0,Y 573.077,Z 372.44,A -85,B 0,C 180,E1 -2100.858,E2 -2100.858} C_VEL
LIN {X 0,Y 573.01,Z 375.493,A -85,B 0,C 180,E1 -2103.495,E2 -2103.495} C_VEL
LIN {X 0,Y 573.028,Z 378.521,A -85,B 0,C 180,E1 -2106.061,E2 -2106.061} C_VEL
LIN {X 0,Y 572.983,Z 381.552,A -85,B 0,C 180,E1 -2108.718,E2 -2108.718} C_VEL
LIN {X 0,Y 572.979,Z 385.166,A -85,B 0,C 180,E1 -2111.566,E2 -2111.566} C_VEL
LIN {X 0,Y 572.974,Z 389.156,A -85,B 0,C 180,E1 -2114.651,E2 -2114.651} C_VEL
LIN {X 0,Y 572.98,Z 393.003,A -85,B 0,C 180,E1 -2117.577,E2 -2117.577} C_VEL
LIN {X 0,Y 572.932,Z 395.682,A -85,B 0,C 180,E1 -2119.59,E2 -2119.59} C_VEL
LIN {X 0,Y 573.833,Z 402.644,A -85,B 0,C 180,E1 -2119.766,E2 -2119.766} C_VEL
LIN {X 0,Y 573.716,Z 415.414,A -85,B 0,C 180,E1 -2120.148,E2 -2120.148} C_VEL
LIN {X 0,Y 573.61,Z 427.432,A -85,B 0,C 180,E1 -2120.651,E2 -2120.651} C_VEL
LIN {X 0,Y 573.486,Z 439.475,A -85,B 0,C 180,E1 -2121.319,E2 -2121.319} C_VEL
LIN {X 0,Y 573.386,Z 450.669,A -85,B 0,C 180,E1 -2122.107,E2 -2122.107} C_VEL
LIN {X 0,Y 573.284,Z 460.328,A -85,B 0,C 180,E1 -2122.952,E2 -2122.952} C_VEL
LIN {X 0,Y 573.162,Z 470.147,A -85,B 0,C 180,E1 -2124.019,E2 -2124.019} C_VEL
LIN {X 0,Y 573.083,Z 477.809,A -85,B 0,C 180,E1 -2125.051,E2 -2125.051} C_VEL
LIN {X 0,Y 573.057,Z 485.061,A -85,B 0,C 180,E1 -2126.294,E2 -2126.294} C_VEL
LIN {X 0,Y 573.004,Z 489.838,A -85,B 0,C 180,E1 -2127.34,E2 -2127.34} C_VEL
LIN {X 0,Y 572.99,Z 494.119,A -85,B 0,C 180,E1 -2128.583,E2 -2128.583} C_VEL
LIN {X 0,Y 572.942,Z 496.989,A -85,B 0,C 180,E1 -2129.807,E2 -2129.807} C_VEL
LIN {X 0,Y 572.965,Z 498.163,A -85,B 0,C 180,E1 -2130.618,E2 -2130.618} C_VEL
LIN {X 0,Y 572.92,Z 498.999,A -85,B 0,C 180,E1 -2132.025,E2 -2132.025} C_VEL
LIN {X 0,Y 572.931,Z 498.61,A -85,B 0,C 180,E1 -2133.009,E2 -2133.009} C_VEL
LIN {X 0,Y 572.943,Z 497.764,A -85,B 0,C 180,E1 -2133.795,E2 -2133.795} C_VEL
LIN {X 0,Y 572.964,Z 495.006,A -85,B 0,C 180,E1 -2135.177,E2 -2135.177} C_VEL
LIN {X 0,Y 573.021,Z 490.804,A -85,B 0,C 180,E1 -2136.51,E2 -2136.51} C_VEL
LIN {X 0,Y 573.028,Z 485.789,A -85,B 0,C 180,E1 -2137.654,E2 -2137.654} C_VEL
LIN {X 0,Y 573.082,Z 479.703,A -85,B 0,C 180,E1 -2138.741,E2 -2138.741} C_VEL
LIN {X 0,Y 573.153,Z 472.82,A -85,B 0,C 180,E1 -2139.733,E2 -2139.733} C_VEL
LIN {X 0,Y 573.231,Z 463.546,A -85,B 0,C 180,E1 -2140.817,E2 -2140.817} C_VEL
LIN {X 0,Y 573.353,Z 454.184,A -85,B 0,C 180,E1 -2141.694,E2 -2141.694} C_VEL
LIN {X 0,Y 573.411,Z 443.251,A -85,B 0,C 180,E1 -2142.526,E2 -2142.526} C_VEL
LIN {X 0,Y 573.541,Z 432.527,A -85,B 0,C 180,E1 -2143.178,E2 -2143.178} C_VEL
LIN {X 0,Y 573.67,Z 421.011,A -85,B 0,C 180,E1 -2143.726,E2 -2143.726} C_VEL
LIN {X 0,Y 573.805,Z 407.829,A -85,B 0,C 180,E1 -2144.187,E2 -2144.187} C_VEL
LIN {X 0,Y 573.659,Z 400.214,A -85,B 0,C 180,E1 -2144.387,E2 -2144.387} C_VEL
LIN {X 0,Y 572.961,Z 395.674,A -85,B 0,C 180,E1 -2144.505,E2 -2144.505} C_VEL
LIN {X 0,Y 572.931,Z 392.038,A -85,B 0,C 180,E1 -2147.245,E2 -2147.245} C_VEL
LIN {X 0,Y 572.953,Z 389.21,A -85,B 0,C 180,E1 -2149.398,E2 -2149.398} C_VEL
LIN {X 0,Y 572.953,Z 385.523,A -85,B 0,C 180,E1 -2152.246,E2 -2152.246} C_VEL
LIN {X 0,Y 572.973,Z 381.926,A -85,B 0,C 180,E1 -2155.075,E2 -2155.075} C_VEL
LIN {X 0,Y 572.977,Z 379.612,A -85,B 0,C 180,E1 -2157.188,E2 -2157.188} C_VEL
LIN {X 0,Y 573.111,Z 377.437,A -85,B 0,C 180,E1 -2159.298,E2 -2159.298} C_VEL
LIN {X 0,Y 573.117,Z 374.973,A -85,B 0,C 180,E1 -2161.406,E2 -2161.406} C_VEL
LIN {X 0,Y 573.153,Z 371.744,A -85,B 0,C 180,E1 -2164.22,E2 -2164.22} C_VEL
LIN {X 0,Y 573.168,Z 369.302,A -85,B 0,C 180,E1 -2166.336,E2 -2166.336} C_VEL
LIN {X 0,Y 573.274,Z 369.077,A -85,B 0,C 180,E1 -2168.46,E2 -2168.46} C_VEL
LIN {X 0,Y 573.288,Z 369.074,A -85,B 0,C 180,E1 -2171.312,E2 -2171.312} C_VEL
LIN {X 0,Y 573.244,Z 369.08,A -85,B 0,C 180,E1 -2174.427,E2 -2174.427} C_VEL
LIN {X 0,Y 573.267,Z 369.076,A -85,B 0,C 180,E1 -2177.112,E2 -2177.112} C_VEL
LIN {X 0,Y 573.232,Z 369.08,A -85,B 0,C 180,E1 -2180.078,E2 -2180.078} C_VEL
LIN {X 0,Y 573.275,Z 369.075,A -85,B 0,C 180,E1 -2183.165,E2 -2183.165} C_VEL
LIN {X 0,Y 573.257,Z 369.078,A -85,B 0,C 180,E1 -2186.191,E2 -2186.191} C_VEL
LIN {X 0,Y 573.229,Z 369.081,A -85,B 0,C 180,E1 -2188.565,E2 -2188.565} C_VEL
LIN {X 0,Y 573.215,Z 369.087,A -85,B 0,C 180,E1 -2190.994,E2 -2190.994} C_VEL
LIN {X 0,Y 573.258,Z 369.077,A -85,B 0,C 180,E1 -2193.531,E2 -2193.531} C_VEL
LIN {X 0,Y 573.25,Z 369.078,A -85,B 0,C 180,E1 -2196.049,E2 -2196.049} C_VEL
LIN {X 0,Y 573.225,Z 369.084,A -85,B 0,C 180,E1 -2198.704,E2 -2198.704} C_VEL
LIN {X 0,Y 573.243,Z 369.082,A -85,B 0,C 180,E1 -2201.6,E2 -2201.6} C_VEL
LIN {X 0,Y 573.215,Z 369.087,A -85,B 0,C 180,E1 -2204.336,E2 -2204.336} C_VEL
LIN {X 0,Y 573.24,Z 369.084,A -85,B 0,C 180,E1 -2207.359,E2 -2207.359} C_VEL
LIN {X 0,Y 573.229,Z 369.087,A -85,B 0,C 180,E1 -2210.396,E2 -2210.396} C_VEL
LIN {X 0,Y 573.284,Z 369.19,A -85,B 0,C 180,E1 -2213.194,E2 -2213.194} C_VEL
LIN {X 0,Y 573.792,Z 373.804,A -85,B 0,C 180,E1 -2214.858,E2 -2214.858} C_VEL
LIN {X 0,Y 573.64,Z 381.432,A -85,B 0,C 180,E1 -2217.384,E2 -2217.384} C_VEL
LIN {X 0,Y 573.528,Z 391.516,A -85,B 0,C 180,E1 -2220.463,E2 -2220.463} C_VEL
LIN {X 0,Y 573.438,Z 401.744,A -85,B 0,C 180,E1 -2223.468,E2 -2223.468} C_VEL
LIN {X 0,Y 573.389,Z 410.998,A -85,B 0,C 180,E1 -2226.145,E2 -2226.145} C_VEL
LIN {X 0,Y 573.263,Z 419.935,A -85,B 0,C 180,E1 -2228.707,E2 -2228.707} C_VEL
LIN {X 0,Y 573.213,Z 429.532,A -85,B 0,C 180,E1 -2231.414,E2 -2231.414} C_VEL
LIN {X 0,Y 573.16,Z 440.123,A -85,B 0,C 180,E1 -2234.353,E2 -2234.353} C_VEL
LIN {X 0,Y 573.098,Z 449.39,A -85,B 0,C 180,E1 -2236.89,E2 -2236.89} C_VEL
LIN {X 0,Y 573.085,Z 451.541,A -85,B 0,C 180,E1 -2237.475,E2 -2237.475} C_VEL
LIN {X 0,Y 573.874,Z 457.384,A -85,B 0,C 180,E1 -2237.605,E2 -2237.605} C_VEL
LIN {X 0,Y 573.79,Z 470.6,A -85,B 0,C 180,E1 -2237.94,E2 -2237.94} C_VEL
LIN {X 0,Y 573.65,Z 482.814,A -85,B 0,C 180,E1 -2238.396,E2 -2238.396} C_VEL
LIN {X 0,Y 573.523,Z 494.472,A -85,B 0,C 180,E1 -2238.976,E2 -2238.976} C_VEL
LIN {X 0,Y 573.451,Z 505.523,A -85,B 0,C 180,E1 -2239.678,E2 -2239.678} C_VEL
LIN {X 0,Y 573.306,Z 515.68,A -85,B 0,C 180,E1 -2240.477,E2 -2240.477} C_VEL
LIN {X 0,Y 573.214,Z 524.813,A -85,B 0,C 180,E1 -2241.365,E2 -2241.365} C_VEL
LIN {X 0,Y 573.14,Z 533.711,A -85,B 0,C 180,E1 -2242.428,E2 -2242.428} C_VEL
LIN {X 0,Y 573.049,Z 540.416,A -85,B 0,C 180,E1 -2243.417,E2 -2243.417} C_VEL
LIN {X 0,Y 573.07,Z 545.694,A -85,B 0,C 180,E1 -2244.372,E2 -2244.372} C_VEL
LIN {X 0,Y 573.028,Z 550.383,A -85,B 0,C 180,E1 -2245.43,E2 -2245.43} C_VEL
LIN {X 0,Y 573.022,Z 553.965,A -85,B 0,C 180,E1 -2246.487,E2 -2246.487} C_VEL
LIN {X 0,Y 572.959,Z 555.815,A -85,B 0,C 180,E1 -2247.19,E2 -2247.19} C_VEL
LIN {X 0,Y 572.939,Z 557.203,A -85,B 0,C 180,E1 -2247.894,E2 -2247.894} C_VEL
LIN {X 0,Y 572.94,Z 558.786,A -85,B 0,C 180,E1 -2249.3,E2 -2249.3} C_VEL
LIN {X 0,Y 572.938,Z 559,A -85,B 0,C 180,E1 -2250.003,E2 -2250.003} C_VEL
LIN {X 0,Y 572.946,Z 558.183,A -85,B 0,C 180,E1 -2251.408,E2 -2251.408} C_VEL
LIN {X 0,Y 572.94,Z 557.196,A -85,B 0,C 180,E1 -2252.111,E2 -2252.111} C_VEL
LIN {X 0,Y 572.959,Z 555.804,A -85,B 0,C 180,E1 -2252.815,E2 -2252.815} C_VEL
LIN {X 0,Y 573.015,Z 552.888,A -85,B 0,C 180,E1 -2253.87,E2 -2253.87} C_VEL
LIN {X 0,Y 572.963,Z 548.939,A -85,B 0,C 180,E1 -2254.928,E2 -2254.928} C_VEL
LIN {X 0,Y 573.069,Z 542.863,A -85,B 0,C 180,E1 -2256.163,E2 -2256.163} C_VEL
LIN {X 0,Y 573.122,Z 536.221,A -85,B 0,C 180,E1 -2257.223,E2 -2257.223} C_VEL
LIN {X 0,Y 573.193,Z 527.971,A -85,B 0,C 180,E1 -2258.286,E2 -2258.286} C_VEL
LIN {X 0,Y 573.288,Z 519.514,A -85,B 0,C 180,E1 -2259.173,E2 -2259.173} C_VEL
LIN {X 0,Y 573.418,Z 509.067,A -85,B 0,C 180,E1 -2260.061,E2 -2260.061} C_VEL
LIN {X 0,Y 573.516,Z 497.498,A -85,B 0,C 180,E1 -2260.849,E2 -2260.849} C_VEL
LIN {X 0,Y 573.616,Z 485.833,A -85,B 0,C 180,E1 -2261.468,E2 -2261.468} C_VEL
LIN {X 0,Y 573.753,Z 473.108,A -85,B 0,C 180,E1 -2261.976,E2 -2261.976} C_VEL
LIN {X 0,Y 573.872,Z 460.427,A -85,B 0,C 180,E1 -2262.333,E2 -2262.333} C_VEL
LIN {X 0,Y 573.572,Z 454.682,A -85,B 0,C 180,E1 -2262.454,E2 -2262.454} C_VEL
LIN {X 0,Y 573.088,Z 451.522,A -85,B 0,C 180,E1 -2262.53,E2 -2262.53} C_VEL
LIN {X 0,Y 573.16,Z 441.428,A -85,B 0,C 180,E1 -2265.288,E2 -2265.288} C_VEL
LIN {X 0,Y 573.219,Z 430.837,A -85,B 0,C 180,E1 -2268.221,E2 -2268.221} C_VEL
LIN {X 0,Y 573.297,Z 421.57,A -85,B 0,C 180,E1 -2270.827,E2 -2270.827} C_VEL
LIN {X 0,Y 573.357,Z 412.304,A -85,B 0,C 180,E1 -2273.478,E2 -2273.478} C_VEL
LIN {X 0,Y 573.424,Z 402.96,A -85,B 0,C 180,E1 -2276.184,E2 -2276.184} C_VEL
LIN {X 0,Y 573.48,Z 393.537,A -85,B 0,C 180,E1 -2278.954,E2 -2278.954} C_VEL
LIN {X 0,Y 573.611,Z 385.581,A -85,B 0,C 180,E1 -2281.382,E2 -2281.382} C_VEL
LIN {X 0,Y 573.753,Z 376.395,A -85,B 0,C 180,E1 -2284.297,E2 -2284.297} C_VEL
LIN {X 0,Y 573.61,Z 371.23,A -85,B 0,C 180,E1 -2286.036,E2 -2286.036} C_VEL
LIN {X 0,Y 573.254,Z 369.082,A -85,B 0,C 180,E1 -2286.814,E2 -2286.814} C_VEL
LIN {X 0,Y 573.247,Z 369.081,A -85,B 0,C 180,E1 -2289.609,E2 -2289.609} C_VEL
LIN {X 0,Y 573.232,Z 369.081,A -85,B 0,C 180,E1 -2292.64,E2 -2292.64} C_VEL
LIN {X 0,Y 573.218,Z 369.082,A -85,B 0,C 180,E1 -2295.328,E2 -2295.328} C_VEL
LIN {X 0,Y 573.234,Z 369.083,A -85,B 0,C 180,E1 -2298.408,E2 -2298.408} C_VEL
LIN {X 0,Y 573.243,Z 369.084,A -85,B 0,C 180,E1 -2301.298,E2 -2301.298} C_VEL
LIN {X 0,Y 573.199,Z 369.088,A -85,B 0,C 180,E1 -2304.022,E2 -2304.022} C_VEL
LIN {X 0,Y 573.242,Z 369.082,A -85,B 0,C 180,E1 -2306.516,E2 -2306.516} C_VEL
LIN {X 0,Y 573.228,Z 369.084,A -85,B 0,C 180,E1 -2309.12,E2 -2309.12} C_VEL
LIN {X 0,Y 573.236,Z 369.08,A -85,B 0,C 180,E1 -2311.435,E2 -2311.435} C_VEL
LIN {X 0,Y 573.247,Z 369.082,A -85,B 0,C 180,E1 -2314.589,E2 -2314.589} C_VEL
LIN {X 0,Y 573.246,Z 369.08,A -85,B 0,C 180,E1 -2316.901,E2 -2316.901} C_VEL
LIN {X 0,Y 573.258,Z 369.078,A -85,B 0,C 180,E1 -2319.173,E2 -2319.173} C_VEL
LIN {X 0,Y 573.222,Z 369.086,A -85,B 0,C 180,E1 -2321.411,E2 -2321.411} C_VEL
LIN {X 0,Y 573.253,Z 369.079,A -85,B 0,C 180,E1 -2323.621,E2 -2323.621} C_VEL
LIN {X 0,Y 573.225,Z 369.083,A -85,B 0,C 180,E1 -2326.529,E2 -2326.529} C_VEL
LIN {X 0,Y 573.272,Z 369.076,A -85,B 0,C 180,E1 -2328.745,E2 -2328.745} C_VEL
LIN {X 0,Y 573.261,Z 369.077,A -85,B 0,C 180,E1 -2331.54,E2 -2331.54} C_VEL
LIN {X 0,Y 573.237,Z 369.082,A -85,B 0,C 180,E1 -2333.664,E2 -2333.664} C_VEL
